(* IEC 61131-3 sources: TSA-FMICS22/benchmark/PLCopen_safety/examples, 5 files *)

(* ---- 4.1.DiagnosticsConcept.st ---- *)
PROGRAM DiagnosticsConcept
VAR_INPUT
    S1SEStopIn1 : SAFEBOOL;
    S1SEStopIn2 : SAFEBOOL;
    S2SESPEIn : SAFEBOOL;
    S0Reset : BOOL;
    S3DriveReset : BOOL;
    AxisD1 : INT;
    InputDevice1active : BOOL;
    InputDevice2active : BOOL;
    InternalAcknowledge: BOOL;
END_VAR
VAR
    SEStopOut : SAFEBOOL;
    SFEquivalent1 : SFEquivalent;
    SFEmergencyStop1 : SFEmergencyStop;
    SFESPE1 : SFESPE;
    SFSafeStop11 : SFSafeStop;
END_VAR
VAR_OUTPUT
    ErrorEquiv1 : BOOL;
    DiagEquiv1 : WORD;
    ErrorEStop1 : BOOL;
    DiagEStop1 : WORD;
    ErrorESPE1 : BOOL;
    DiagESPE1 : WORD;
    ErrorSafeStop1 : BOOL;
    DiagSafeStop1 : WORD;
    SStopped : BOOL;
END_VAR
SFEquivalent1(Activate:=InputDevice1active, SChannelA:=S1SEStopIn1, SChannelB:=S1SEStopIn2, DiscrepancyTime:=T#10ms);
SFEmergencyStop1(Activate:=SFEquivalent1.Ready, SEStopIn:=SFEquivalent1.SEquivalentOut, SStartReset:=FALSE, SAutoReset:=FALSE, Reset:=S0Reset);
SFESPE1(Activate:=InputDevice2active, SESPEIn:=S2SESPEIn, SStartReset:=FALSE, SAutoReset:=FALSE, Reset:=S0Reset);
SFSafeStop11(Activate:=SFEmergencyStop1.Ready AND SFESPE1.Ready, SStopIn:=SEStopOut AND SFESPE1.SESPEOut, AxisID:=AxisD1, MonitoringTime:=T#100ms, Reset:=S3DriveReset, Acknowledge := InternalAcknowledge);
SEStopOut := SFEmergencyStop1.SEStopOut;
ErrorEquiv1 := SFEquivalent1.Error;
DiagEquiv1 := SFEquivalent1.DiagCode;
ErrorEStop1 := SFEmergencyStop1.Error;
DiagEStop1 := SFEmergencyStop1.DiagCode;
ErrorESPE1 := SFESPE1.Error;
DiagESPE1 := SFESPE1.DiagCode;
ErrorSafeStop1 := SFSafeStop11.Error;
DiagSafeStop1 := SFSafeStop11.DiagCode;
SStopped := SFSafeStop11.SStopped;
END_PROGRAM

FUNCTION_BLOCK SFEquivalent
VAR_INPUT
    Activate : BOOL;
    SChannelA : BOOL;
    SChannelB : BOOL;
    DiscrepancyTime : TIME;
END_VAR
VAR
    Timer : TON;
END_VAR
VAR_OUTPUT
    Ready : BOOL;
	SEquivalentOut : BOOL;
	Error : BOOL;
	DiagCode : WORD;
END_VAR

IF NOT Activate THEN
    DiagCode := 16#0000;
ELSE
    CASE DiagCode OF
    16#0000:
        IF Activate THEN
            DiagCode := 16#8001;
        END_IF;
    16#8001:
        IF SChannelA AND NOT SChannelB THEN
            DiagCode := 16#8004;
        ELSIF SChannelB AND NOT SChannelA THEN
            DiagCode := 16#8014;
        ELSIF SChannelA AND SChannelB THEN
            DiagCode := 16#8000;
        END_IF;
    16#8004:
        IF Timer.Q THEN
            DiagCode := 16#C001;
        ELSIF NOT SChannelA THEN
            DiagCode := 16#8001;
        ELSIF SChannelB THEN
            DiagCode := 16#8000;
        END_IF;
    16#C001,
    16#C002:
        IF NOT SChannelA AND NOT SChannelB THEN
            DiagCode := 16#8001;
        END_IF;
    16#8014:
        IF Timer.Q THEN
            DiagCode := 16#C002;
        ELSIF NOT SChannelB THEN
            DiagCode := 16#8001;
        ELSIF SChannelA THEN
            DiagCode := 16#8000;
        END_IF;
    16#C003:
        IF NOT SChannelA AND NOT SChannelB THEN
            DiagCode := 16#8001;
        END_IF;
    16#8005:
        IF Timer.Q THEN
            DiagCode := 16#C003;
        ELSIF NOT SChannelA AND NOT SChannelB THEN
            DiagCode := 16#8001;
        END_IF;
    16#8000:
        IF SChannelA XOR SChannelB THEN
            DiagCode := 16#8005;
        ELSIF NOT SChannelA AND NOT SChannelB THEN
            DiagCode := 16#8001;
        END_IF;
    END_CASE;
END_IF;

CASE DiagCode OF
16#0000:
    Timer(IN:=FALSE, PT:=DiscrepancyTime);
    Ready := FALSE;
    Error := FALSE;
    SEquivalentOut:= FALSE;
16#8000:
    Timer(IN:=FALSE, PT:=DiscrepancyTime);
    Ready := TRUE;
    Error := FALSE;
    SEquivalentOut := TRUE;
16#8001:
    Timer(IN:=FALSE, PT:=DiscrepancyTime);
    Ready := TRUE;
    Error := FALSE;
    SEquivalentOut:= FALSE;
16#8004,
16#8014,
16#8005:
	Timer(IN:=TRUE, PT:=DiscrepancyTime);
    Ready := TRUE;
    Error := FALSE;
    SEquivalentOut:= FALSE;
16#C001,
16#C002,
16#C003:
    Timer(IN:=FALSE, PT:=DiscrepancyTime);
    Ready := TRUE;
    Error := TRUE;
    SEquivalentOut:= FALSE;
END_CASE;
END_FUNCTION_BLOCK

FUNCTION_BLOCK SFEmergencyStop
VAR_INPUT
    Activate : BOOL;
    SEStopIn : BOOL;
    SStartReset : BOOL;
    SAutoReset : BOOL;
    Reset : BOOL;
END_VAR
VAR
    RTRIGatReset : RTRIG;
END_VAR
VAR_OUTPUT
    Ready : BOOL;
    SEStopOut : BOOL;
    Error : BOOL;
    DiagCode : WORD;
END_VAR
RTRIGatReset(CLK:=Reset);
IF NOT Activate THEN
    DiagCode := 16#0000;
ELSE
    CASE DiagCode OF
    16#0000:
        IF Activate THEN
            DiagCode := 16#8001;
        END_IF;
    16#8001:
        IF NOT SStartReset THEN
            DiagCode := 16#8002;
        ELSIF SStartReset AND NOT SEStopIn THEN
            DiagCode := 16#8004;
        ELSIF SEStopIn AND SStartReset THEN
            DiagCode := 16#8000;
        END_IF;
    16#8002:
        IF SEStopIn THEN
            DiagCode := 16#8003;
        END_IF;
    16#8003:
        IF Reset AND NOT RTRIGatReset.Q THEN
            DiagCode := 16#C001;
        ELSIF NOT SEStopIn THEN
            DiagCode := 16#8002;
        ELSIF RTRIGatReset.Q THEN
            DiagCode := 16#8000;
        END_IF;
    16#C001:
        IF NOT Reset THEN
            DiagCode := 16#8003;
        END_IF;
    16#8004:
        IF SEStopIn AND NOT SAutoReset THEN
            DiagCode := 16#8005;
        ELSIF SEStopIn AND SAutoReset THEN
            DiagCode := 16#8000;
        END_IF;
    16#8005:
        IF Reset AND NOT RTRIGatReset.Q THEN
            DiagCode := 16#C002;
        ELSIF NOT SEStopIn THEN
            DiagCode := 16#8004;
        ELSIF RTRIGatReset.Q OR SAutoReset THEN
            DiagCode := 16#8000;
        END_IF;
    16#C002:
        IF NOT Reset THEN
            DiagCode := 16#8005;
        END_IF;
    16#8000:
        IF NOT SEStopIn THEN
            DiagCode := 16#8004;
        END_IF;
    END_CASE;
END_IF;
CASE DiagCode OF
16#0000:
    Ready := FALSE;
    Error := FALSE;
    SEStopOut := FALSE;
16#8001:
    Ready := TRUE;
    Error := FALSE;
    SEStopOut := FALSE;
16#8002:
    Ready := TRUE;
    Error := FALSE;
    SEStopOut := FALSE;
16#8003:
    Ready := TRUE;
    Error := FALSE;
    SEStopOut := FALSE;
16#C001:
    Ready := TRUE;
    Error := TRUE;
    SEStopOut := FALSE;
16#8004:
    Ready := TRUE;
    Error := FALSE;
    SEStopOut := FALSE;
16#8005:
    Ready := TRUE;
    Error := FALSE;
    SEStopOut := FALSE;
16#C002:
    Ready := TRUE;
    Error := TRUE;
    SEStopOut := FALSE;
16#8000:
    Ready := TRUE;
    Error := FALSE;
    SEStopOut := TRUE;
END_CASE;
END_FUNCTION_BLOCK

FUNCTION_BLOCK SFESPE
VAR_INPUT
    Activate : BOOL;
    SESPEIn : BOOL;
    SStartReset : BOOL;
    SAutoReset : BOOL;
    Reset : BOOL;
END_VAR
VAR
    RTRIGatReset : RTRIG;
END_VAR
VAR_OUTPUT
    Ready : BOOL;
    SESPEOut : BOOL;
    Error : BOOL;
    DiagCode : WORD;
END_VAR
RTRIGatReset(CLK:=Reset);
IF NOT Activate THEN
    DiagCode := 16#0000;
ELSE
    CASE DiagCode OF
    16#0000:
        IF Activate THEN
            DiagCode := 16#8001;
        END_IF;
    16#8001:
        IF NOT SStartReset THEN
            DiagCode := 16#8002;
        ELSIF SStartReset AND NOT SESPEIn THEN
            DiagCode := 16#8004;
        ELSIF SESPEIn AND SStartReset THEN
            DiagCode := 16#8000;
        END_IF;
    16#8002:
        IF SESPEIn THEN
            DiagCode := 16#8003;
        END_IF;
    16#8003:
        IF Reset AND NOT RTRIGatReset.Q THEN
            DiagCode := 16#C001;
        ELSIF NOT SESPEIn THEN
            DiagCode := 16#8002;
        ELSIF RTRIGatReset.Q THEN
            DiagCode := 16#8000;
        END_IF;
    16#C001:
        IF NOT Reset THEN
            DiagCode := 16#8003;
        END_IF;
    16#8004:
        IF SESPEIn AND NOT SAutoReset THEN
            DiagCode := 16#8005;
        ELSIF SESPEIn AND SAutoReset THEN
            DiagCode := 16#8000;
        END_IF;
    16#8005:
        IF Reset AND NOT RTRIGatReset.Q THEN
            DiagCode := 16#C002;
        ELSIF NOT SESPEIn THEN
            DiagCode := 16#8004;
        ELSIF RTRIGatReset.Q OR SAutoReset THEN
            DiagCode := 16#8000;
        END_IF;
    16#C002:
        IF NOT Reset THEN
            DiagCode := 16#8005;
        END_IF;
    16#8000:
        IF NOT SESPEIn THEN
            DiagCode := 16#8004;
        END_IF;
    END_CASE;
END_IF;
CASE DiagCode OF
16#0000:
    Ready := FALSE;
    Error := FALSE;
    SESPEOut := FALSE;
16#8001:
    Ready := TRUE;
    Error := FALSE;
    SESPEOut := FALSE;
16#8002:
    Ready := TRUE;
    Error := FALSE;
    SESPEOut := FALSE;
16#8003:
    Ready := TRUE;
    Error := FALSE;
    SESPEOut := FALSE;
16#C001:
    Ready := TRUE;
    Error := TRUE;
    SESPEOut := FALSE;
16#8004:
    Ready := TRUE;
    Error := FALSE;
    SESPEOut := FALSE;
16#8005:
    Ready := TRUE;
    Error := FALSE;
    SESPEOut := FALSE;
16#C002:
    Ready := TRUE;
    Error := TRUE;
    SESPEOut := FALSE;
16#8000:
    Ready := TRUE;
    Error := FALSE;
    SESPEOut := TRUE;
END_CASE;
END_FUNCTION_BLOCK

FUNCTION_BLOCK SFSafeStop
VAR_INPUT
    Activate : BOOL;
    SStopIn : SAFEBOOL;
    AxisID : INT;
    MonitoringTime : TIME;
    Reset : BOOL;
    Acknowledge : BOOL;      (* This is an internal input *)
END_VAR
VAR
    Timer : TON;
    RTRIGatReset : RTRIG;
END_VAR
VAR_OUTPUT
    Ready : BOOL;
    SStopped : SAFEBOOL;
    Error : BOOL;
    DiagCode : WORD:=16#0000;
END_VAR
RTRIGatReset(CLK:=Reset);
IF NOT Activate THEN
    DiagCode := 16#0000;
ELSE
    Timer(IN:=Activate AND NOT SStopIn, PT:=MonitoringTime);
    CASE DiagCode OF
    16#0000:
        IF Activate THEN
            DiagCode := 16#8001;
        END_IF;
    16#8000:
        IF NOT Acknowledge THEN
            DiagCode := 16#C002;
        ELSIF SStopIn THEN
            DiagCode := 16#8012;
        END_IF;
    16#8001:
        IF RTRIGatReset.Q AND NOT Acknowledge THEN
            DiagCode := 16#8002;
        ELSIF RTRIGatReset.Q AND Acknowledge THEN
            DiagCode := 16#8012;
        END_IF;
    16#8002:
        IF NOT SStopIn THEN
            DiagCode := 16#8003;
        ELSIF Acknowledge THEN
            DiagCode := 16#8012;
        END_IF;
    16#8003:
        IF Timer.Q THEN
            DiagCode := 16#C003;
        ELSIF SStopIn THEN
            DiagCode := 16#8012;
        ELSIF Acknowledge THEN
            DiagCode := 16#8000;
        END_IF;
    16#8005:
        IF SStopIn THEN
            DiagCode := 16#8012;
        END_IF;
    16#8012:
        IF NOT Acknowledge THEN
            DiagCode := 16#8002;
        ELSIF NOT SStopIn THEN
            DiagCode := 16#8003;
        ELSIF Acknowledge THEN
            DiagCode := 16#8000;
        END_IF;
    16#C002:
        IF Reset AND NOT RTRIGatReset.Q THEN
            DiagCode := 16#C004;
        ELSIF RTRIGatReset.Q THEN
            DiagCode := 16#8005;
        END_IF;
    16#C003:
        IF Reset AND NOT RTRIGatReset.Q THEN
            DiagCode := 16#C005;
        ELSIF RTRIGatReset.Q THEN
            DiagCode := 16#8005;
        END_IF;
    16#C004:
        IF NOT Reset THEN
            DiagCode := 16#C002;
        END_IF;
    16#C005:
        IF NOT Reset THEN
            DiagCode := 16#C003;
        END_IF;
    END_CASE;
END_IF;
CASE DiagCode OF
16#0000:
    Ready := FALSE;
    SStopped := FALSE;
    Error := FALSE;
16#8000:
    Ready := TRUE;
    SStopped := TRUE;
    Error := FALSE;
16#8001,
16#8002,
16#8003,
16#8005,
16#8012:
    Ready := TRUE;
    SStopped := FALSE;
    Error := FALSE;
16#C002,
16#C003,
16#C004,
16#C005:
    Ready := TRUE;
    SStopped := FALSE;
    Error := TRUE;
END_CASE;
END_FUNCTION_BLOCK

FUNCTION_BLOCK RTRIG
VAR_INPUT
    CLK : BOOL;
END_VAR
VAR
    M : BOOL;
END_VAR
VAR_OUTPUT
    Q : BOOL;
END_VAR
    Q := CLK AND NOT M;
    M := CLK;
END_FUNCTION_BLOCK

FUNCTION_BLOCK TON
VAR_INPUT
    IN : BOOL;
    PT : TIME;
END_VAR
VAR
    running : BOOL;
END_VAR
VAR_TEMP
    timeout : BOOL;
END_VAR
VAR_OUTPUT
    Q : BOOL;
    ET : TIME;
END_VAR
timeout := NONDETERMINISTIC_BOOL();
IF NOT IN THEN
    Q := FALSE;
    running := FALSE;
ELSIF NOT running AND NOT Q THEN
    running := TRUE;
ELSIF running AND NOT Q THEN
    Q := timeout;
    running := NOT Q;
END_IF;
ET := NONDETERMINISTIC_TIME();
END_FUNCTION_BLOCK

(* ---- 4.2.SafeMotion.st ---- *)
PROGRAM SafeMotion
VAR_INPUT
    S1SEStopIn : SAFEBOOL;
    S2SMode0 : SAFEBOOL;
    S2SMode1 : SAFEBOOL;
    S4SEnableSwitchCh1 : SAFEBOOL;
    S4SEnableSwitchCh2 : SAFEBOOL;
    S5SGuardSwitch1 : SAFEBOOL;
    S6SGuardSwitch2 : SAFEBOOL;
    S7SGuardLock : SAFEBOOL;
    S0Reset : BOOL;
    S8UnlockGuard : BOOL;
    SFSafeStop11ACK: BOOL;
    SFSafeStop12ACK: BOOL;
    SFSLS1ACK: BOOL;
    SFSLS2ACK: BOOL;
END_VAR
VAR_OUTPUT
    SUnlockGuardK1 : SAFEBOOL;
END_VAR
VAR
    SSafeStopAxis1 : SAFEBOOL;
    SSafeStopAxis2 : SAFEBOOL;
    SSafeMoveAxis1 : SAFEBOOL;
    SSafeMoveAxis2 : SAFEBOOL;
    SSafetyActive : SAFEBOOL;
    SModeAutoActive : SAFEBOOL;
    SModeSetSel : SAFEBOOL;
    SSLSEnable : SAFEBOOL;
    SGuardLocked : SAFEBOOL;
    SFEmergencyStop1 : SFEmergencyStop;
    SFSafeStop11 : SFSafeStop;
    SFSafeStop12 : SFSafeStop;
    SFModeSelector1 : SFModeSelector;
    SFGuardMonitoring1 : SFGuardMonitoring;
    SFGuardLocking1 : SFGuardLocking;
    SFEnableSwitch1 : SFEnableSwitch;
    SFSafelyLimitedSpeed1 : SFSafelyLimitSpeed;
    SFSafelyLimitedSpeed2 : SFSafelyLimitSpeed;
END_VAR

SFEmergencyStop1(Activate:=TRUE, SEStopIn:=S1SEStopIn, SStartReset:=FALSE, SAutoReset:=FALSE, Reset:=S0Reset);
SFSafeStop11(Activate:=TRUE, SStopIn:=SFEmergencyStop1.SEStopOut, AxisID:=1, MonitoringTime:=T#1s, Reset:=S0Reset, Acknowledge:=SFSafeStop11ACK);
SSafeStopAxis1 := SFSafeStop11.SStopped;
SFSafeStop12(Activate:=TRUE, SStopIn:=SFEmergencyStop1.SEStopOut, AxisID:=2, MonitoringTime:=T#1s, Reset:=S0Reset, Acknowledge:=SFSafeStop12ACK);
SSafeStopAxis2 := SFSafeStop12.SStopped;

SFModeSelector1(Activate:=TRUE, SMode0:=S2SMode0, SMode1:=S2SMode1, SMode2:=FALSE, SMode3:=FALSE, SMode4:=FALSE, SMode5:=FALSE, SMode6:=FALSE, SMode7:=FALSE, SUnlock:=TRUE, SSetMode:=FALSE,
 AutoSetMode:=TRUE, ModeMonitorTime:=T#50ms, Reset:=S0Reset);
SModeSetSel := SFModeSelector1.SMode1Sel;
SModeAutoActive := SFModeSelector1.SMode0Sel AND SGuardLocked;

SFGuardMonitoring1(Activate:=TRUE, SGuardSwitch1:=S5SGuardSwitch1, SGuardSwitch2:=S6SGuardSwitch2, DiscrepancyTime:=T#50ms, SStartReset:=FALSE, SAutoReset:=FALSE, Reset:=S0Reset);
SSafetyActive := (SSafeStopAxis1 AND SSafeStopAxis2) OR (SFSafelyLimitedSpeed1.SSafetyActive AND SFSafelyLimitedSpeed2.SSafetyActive);

SFGuardLocking1(Activate:=TRUE, SGuardMonitoring:=SFGuardMonitoring1.SGuardMonitoring, SSafetyActive:=SSafetyActive, SGuardLock:=S7SGuardLock, UnlockRequest:=S8UnlockGuard, SStartReset:=FALSE,
 SAutoReset:=FALSE, Reset:=S0Reset);
SGuardLocked := SFGuardLocking1.SGuardLocked;
SUnlockGuardK1 := SFGuardLocking1.SUnlockGuard;

SFEnableSwitch1(Activate:=TRUE, SSafetyActive:=SSafetyActive AND SModeSetSel, SEnableSwitchCh1:=S4SEnableSwitchCh1, SEnableSwitchCh2:=S4SEnableSwitchCh2, SAutoReset:=FALSE, Reset:=S0Reset);
SSLSEnable := SFEnableSwitch1.SEnableSwitchOut;

SFSafelyLimitedSpeed1(Activate:=TRUE, SOpMode:=SFModeSelector1.SMode0Sel AND SGuardLocked, SEnabled:=SSLSEnable, AxisID:=1, MonitoringTime:=T#1s, Reset:=S0Reset, Acknowledge:=SFSLS1ACK);
SSafeMoveAxis1 := SFSafelyLimitedSpeed1.SSafetyActive;

SFSafelyLimitedSpeed2(Activate:=TRUE, SOpMode:=SFModeSelector1.SMode0Sel AND SGuardLocked, SEnabled:=SSLSEnable, AxisID:=2, MonitoringTime:=T#1s, Reset:=S0Reset, Acknowledge:=SFSLS2ACK);
SSafeMoveAxis2 := SFSafelyLimitedSpeed2.SSafetyActive;
END_PROGRAM

FUNCTION_BLOCK SFEmergencyStop
VAR_INPUT
    Activate : BOOL;
    SEStopIn : BOOL;
    SStartReset : BOOL;
    SAutoReset : BOOL;
    Reset : BOOL;
END_VAR
VAR
    RTRIGatReset : RTRIG;
END_VAR
VAR_OUTPUT
    Ready : BOOL;
    SEStopOut : BOOL;
    Error : BOOL;
    DiagCode : WORD;
END_VAR
RTRIGatReset(CLK:=Reset);
IF NOT Activate THEN
    DiagCode := 16#0000;
ELSE
    CASE DiagCode OF
    16#0000:
        IF Activate THEN
            DiagCode := 16#8001;
        END_IF;
    16#8001:
        IF NOT SStartReset THEN
            DiagCode := 16#8002;
        ELSIF SStartReset AND NOT SEStopIn THEN
            DiagCode := 16#8004;
        ELSIF SEStopIn AND SStartReset THEN
            DiagCode := 16#8000;
        END_IF;
    16#8002:
        IF SEStopIn THEN
            DiagCode := 16#8003;
        END_IF;
    16#8003:
        IF Reset AND NOT RTRIGatReset.Q THEN
            DiagCode := 16#C001;
        ELSIF NOT SEStopIn THEN
            DiagCode := 16#8002;
        ELSIF RTRIGatReset.Q THEN
            DiagCode := 16#8000;
        END_IF;
    16#C001:
        IF NOT Reset THEN
            DiagCode := 16#8003;
        END_IF;
    16#8004:
        IF SEStopIn AND NOT SAutoReset THEN
            DiagCode := 16#8005;
        ELSIF SEStopIn AND SAutoReset THEN
            DiagCode := 16#8000;
        END_IF;
    16#8005:
        IF Reset AND NOT RTRIGatReset.Q THEN
            DiagCode := 16#C002;
        ELSIF NOT SEStopIn THEN
            DiagCode := 16#8004;
        ELSIF RTRIGatReset.Q OR SAutoReset THEN
            DiagCode := 16#8000;
        END_IF;
    16#C002:
        IF NOT Reset THEN
            DiagCode := 16#8005;
        END_IF;
    16#8000:
        IF NOT SEStopIn THEN
            DiagCode := 16#8004;
        END_IF;
    END_CASE;
END_IF;
CASE DiagCode OF
16#0000:
    Ready := FALSE;
    Error := FALSE;
    SEStopOut := FALSE;
16#8001:
    Ready := TRUE;
    Error := FALSE;
    SEStopOut := FALSE;
16#8002:
    Ready := TRUE;
    Error := FALSE;
    SEStopOut := FALSE;
16#8003:
    Ready := TRUE;
    Error := FALSE;
    SEStopOut := FALSE;
16#C001:
    Ready := TRUE;
    Error := TRUE;
    SEStopOut := FALSE;
16#8004:
    Ready := TRUE;
    Error := FALSE;
    SEStopOut := FALSE;
16#8005:
    Ready := TRUE;
    Error := FALSE;
    SEStopOut := FALSE;
16#C002:
    Ready := TRUE;
    Error := TRUE;
    SEStopOut := FALSE;
16#8000:
    Ready := TRUE;
    Error := FALSE;
    SEStopOut := TRUE;
END_CASE;
END_FUNCTION_BLOCK

FUNCTION_BLOCK SFSafeStop
VAR_INPUT
    Activate : BOOL;
    SStopIn : SAFEBOOL;
    AxisID : INT;
    MonitoringTime : TIME;
    Reset : BOOL;
    Acknowledge : BOOL;      (* This is an internal input *)
END_VAR
VAR
    Timer : TON;
    RTRIGatReset : RTRIG;
END_VAR
VAR_OUTPUT
    Ready : BOOL;
    SStopped : SAFEBOOL;
    Error : BOOL;
    DiagCode : WORD:=16#0000;
END_VAR
RTRIGatReset(CLK:=Reset);
IF NOT Activate THEN
    DiagCode := 16#0000;
ELSE
    Timer(IN:=Activate AND NOT SStopIn, PT:=MonitoringTime);
    CASE DiagCode OF
    16#0000:
        IF Activate THEN
            DiagCode := 16#8001;
        END_IF;
    16#8000:
        IF NOT Acknowledge THEN
            DiagCode := 16#C002;
        ELSIF SStopIn THEN
            DiagCode := 16#8012;
        END_IF;
    16#8001:
        IF RTRIGatReset.Q AND NOT Acknowledge THEN
            DiagCode := 16#8002;
        ELSIF RTRIGatReset.Q AND Acknowledge THEN
            DiagCode := 16#8012;
        END_IF;
    16#8002:
        IF NOT SStopIn THEN
            DiagCode := 16#8003;
        ELSIF Acknowledge THEN
            DiagCode := 16#8012;
        END_IF;
    16#8003:
        IF Timer.Q THEN
            DiagCode := 16#C003;
        ELSIF SStopIn THEN
            DiagCode := 16#8012;
        ELSIF Acknowledge THEN
            DiagCode := 16#8000;
        END_IF;
    16#8005:
        IF SStopIn THEN
            DiagCode := 16#8012;
        END_IF;
    16#8012:
        IF NOT Acknowledge THEN
            DiagCode := 16#8002;
        ELSIF NOT SStopIn THEN
            DiagCode := 16#8003;
        ELSIF Acknowledge THEN
            DiagCode := 16#8000;
        END_IF;
    16#C002:
        IF Reset AND NOT RTRIGatReset.Q THEN
            DiagCode := 16#C004;
        ELSIF RTRIGatReset.Q THEN
            DiagCode := 16#8005;
        END_IF;
    16#C003:
        IF Reset AND NOT RTRIGatReset.Q THEN
            DiagCode := 16#C005;
        ELSIF RTRIGatReset.Q THEN
            DiagCode := 16#8005;
        END_IF;
    16#C004:
        IF NOT Reset THEN
            DiagCode := 16#C002;
        END_IF;
    16#C005:
        IF NOT Reset THEN
            DiagCode := 16#C003;
        END_IF;
    END_CASE;
END_IF;
CASE DiagCode OF
16#0000:
    Ready := FALSE;
    SStopped := FALSE;
    Error := FALSE;
16#8000:
    Ready := TRUE;
    SStopped := TRUE;
    Error := FALSE;
16#8001,
16#8002,
16#8003,
16#8005,
16#8012:
    Ready := TRUE;
    SStopped := FALSE;
    Error := FALSE;
16#C002,
16#C003,
16#C004,
16#C005:
    Ready := TRUE;
    SStopped := FALSE;
    Error := TRUE;
END_CASE;
END_FUNCTION_BLOCK

FUNCTION_BLOCK SFModeSelector
VAR_INPUT
    Activate : BOOL;
    SMode0 : BOOL;
    SMode1 : BOOL;
    SMode2 : BOOL;
    SMode3 : BOOL;
    SMode4 : BOOL;
    SMode5 : BOOL;
    SMode6 : BOOL;
    SMode7 : BOOL;
    SUnlock : BOOL;
    SSetMode : BOOL;
    AutoSetMode : BOOL;
    ModeMonitorTime : TIME;
    Reset : BOOL;
END_VAR
VAR
    Timer : TON;
    RTRIGatReset: RTRIG;
    RTRIGatSetMode: RTRIG;
    FTRIGatModeSel0: FTRIG;
    RTRIGatModeSel0: RTRIG;
    fallingEdgeDetected : BOOL;
END_VAR
VAR_TEMP
    Error1 : BOOL;
    Error2 : BOOL;
END_VAR
VAR_OUTPUT
    Ready : BOOL;
    SMode0Sel : BOOL;
    SMode1Sel : BOOL;
    SMode2Sel : BOOL;
    SMode3Sel : BOOL;
    SMode4Sel : BOOL;
    SMode5Sel : BOOL;
    SMode6Sel : BOOL;
    SMode7Sel : BOOL;
    SAnyModeSel : BOOL;
    Error : BOOL;
    DiagCode : WORD;
END_VAR
RTRIGatReset(CLK:=Reset);
RTRIGatSetMode(CLK:=SSetMode);
IF NOT Activate THEN
    DiagCode := 16#0000;
ELSE
    IF (SMode0 + SMode1 + SMode2 + SMode3 + SMode4 + SMode5 + SMode6 + SMode7 > 1) THEN
        Error1 := true;
    ELSE
        Error1 := false;
    END_IF;
    CASE DiagCode OF
    16#0000:
        IF Activate THEN
            DiagCode := 16#8005;
        END_IF;
    16#8005:
        IF (NOT SMode0 AND NOT SMode1 AND NOT SMode2 AND NOT SMode3 AND NOT SMode4 AND NOT SMode5 AND NOT SMode6 AND NOT SMode7) THEN
            FTRIGatModeSel0(CLK:=false);
            RTRIGatModeSel0(CLK:=false);
        ELSE
            FTRIGatModeSel0(CLK:=true);
            RTRIGatModeSel0(CLK:=true);
        END_IF;
        IF FTRIGatModeSel0.Q THEN
            fallingEdgeDetected := TRUE;
        END_IF;
        IF fallingEdgeDetected THEN
            Timer(IN:=TRUE, PT:=ModeMonitorTime);
        ELSIF RTRIGatModeSel0.Q THEN
            Timer(IN:=FALSE, PT:=ModeMonitorTime);
            fallingEdgeDetected := FALSE;
        END_IF;
        Error2 := Timer.Q;
        IF Error1 THEN
            DiagCode := 16#C001;
        ELSIF Error2 THEN
            DiagCode := 16#C002;
        ELSIF ((AutoSetMode OR RTRIGatSetMode.Q) AND SUnlock AND (SMode0 + SMode1 + SMode2 + SMode3 + SMode4 + SMode5 + SMode6 + SMode7 = 1)) THEN
            DiagCode := 16#8000;
        END_IF;
    16#8000:
        IF Error1 THEN
            DiagCode := 16#C001;
        ELSIF (SMode0 <> SMode0Sel OR SMode1 <> SMode1Sel OR SMode2 <> SMode2Sel OR SMode3 <> SMode3Sel
              OR SMode4 <> SMode4Sel OR SMode5 <> SMode5Sel OR SMode6 <> SMode6Sel OR SMode7 <> SMode7Sel) THEN
            DiagCode := 16#8005;
            fallingEdgeDetected := FALSE;
        ELSIF (NOT SUnlock) THEN
            DiagCode := 16#8004;
        END_IF;
    16#8004:
        IF SUnlock THEN
            DiagCode := 16#8000;
        END_IF;
    16#C001:
        IF Reset AND NOT RTRIGatReset.Q THEN
            DiagCode := 16#C003;
        ELSIF RTRIGatReset.Q THEN
            DiagCode := 16#8005;
            fallingEdgeDetected := FALSE;
        END_IF;
    16#C002:
        IF Reset AND NOT RTRIGatReset.Q THEN
            DiagCode := 16#C004;
        ELSIF RTRIGatReset.Q THEN
            DiagCode := 16#8005;
            fallingEdgeDetected := FALSE;
        END_IF;
    16#C003:
        IF (NOT Reset) THEN
            DiagCode := 16#C001;
        END_IF;
    16#C004:
        IF (NOT Reset) THEN
            DiagCode := 16#C002;
        END_IF;
    END_CASE;
END_IF;

CASE DiagCode OF
16#0000:
    Ready := false;
    SMode0Sel := false;
    SMode1Sel := false;
    SMode2Sel := false;
    SMode3Sel := false;
    SMode4Sel := false;
    SMode5Sel := false;
    SMode6Sel := false;
    SMode7Sel := false;
    SAnyModeSel := false;
    Error := false;
16#8005:
    Ready := true;
    SMode0Sel := false;
    SMode1Sel := false;
    SMode2Sel := false;
    SMode3Sel := false;
    SMode4Sel := false;
    SMode5Sel := false;
    SMode6Sel := false;
    SMode7Sel := false;
    SAnyModeSel := false;
    Error := false;
16#8000:
    Ready := true;
    SMode0Sel := SMode0;
    SMode1Sel := SMode1;
    SMode2Sel := SMode2;
    SMode3Sel := SMode3;
    SMode4Sel := SMode4;
    SMode5Sel := SMode5;
    SMode6Sel := SMode6;
    SMode7Sel := SMode7;
    SAnyModeSel := true;
    Error := false;
16#8004:
    Ready := true;
    SAnyModeSel := true;
    Error := false;
16#C001,
16#C002,
16#C003,
16#C004:
    Ready := true;
    SMode0Sel := false;
    SMode1Sel := false;
    SMode2Sel := false;
    SMode3Sel := false;
    SMode4Sel := false;
    SMode5Sel := false;
    SMode6Sel := false;
    SMode7Sel := false;
    SAnyModeSel := false;
    Error := true;
END_CASE;
IF (DiagCode <> 16#8005) THEN
    Timer(IN:=FALSE, PT:=ModeMonitorTime);
END_IF;
END_FUNCTION_BLOCK

FUNCTION_BLOCK SFGuardMonitoring
VAR_INPUT
    Activate : BOOL := FALSE;
    SGuardSwitch1 : SAFEBOOL := FALSE;
    SGuardSwitch2 : SAFEBOOL := FALSE;
    DiscrepancyTime : TIME := T#0s;
    SStartReset : SAFEBOOL := FALSE;
    SAutoReset : SAFEBOOL := FALSE;
    Reset : BOOL := FALSE;
END_VAR
VAR
    Timer : TON;
    RTRIGatReset : RTRIG;
END_VAR
VAR_OUTPUT
    Ready : BOOL := FALSE;
    SGuardMonitoring : BOOL := FALSE;
    Error : BOOL := FALSE;
    DiagCode : WORD := 16#0000;
END_VAR
RTRIGatReset(CLK:=Reset);
IF NOT Activate THEN
    DiagCode := 16#0000;
ELSE
    CASE DiagCode OF
    16#0000:
        IF Activate THEN
            DiagCode := 16#8001;
        END_IF;
    16#8001:
        IF NOT SGuardSwitch1 OR NOT SGuardSwitch2 THEN
            DiagCode := 16#8002;
        ELSIF SGuardSwitch1 AND SGuardSwitch2 AND NOT SStartReset THEN
            DiagCode := 16#8003;
        ELSIF SGuardSwitch1 AND SGuardSwitch2 AND SStartReset THEN
            DiagCode := 16#8000;
        END_IF;
    16#8002:
        IF NOT SGuardSwitch1 AND NOT SGuardSwitch2 THEN
            DiagCode := 16#8012;
        END_IF;
    16#8003:
        IF Reset AND NOT RTRIGatReset.Q THEN
            DiagCode := 16#C001;
        ELSIF NOT SGuardSwitch1 OR NOT SGuardSwitch2 THEN
            DiagCode := 16#8002;
        ELSIF RTRIGatReset.Q THEN
            DiagCode := 16#8000;
        END_IF;
    16#8012:
        IF SGuardSwitch1 THEN
            DiagCode := 16#8004;
        ELSIF SGuardSwitch2 THEN
            DiagCode := 16#8014;
        END_IF;
    16#8004:
        IF Timer.Q THEN
            DiagCode := 16#C011;
        ELSIF NOT SGuardSwitch1 THEN
            DiagCode := 16#8002;
        ELSIF SGuardSwitch2 THEN
            DiagCode := 16#8005;
        END_IF;
    16#8014:
        IF Timer.Q THEN
            DiagCode := 16#C012;
        ELSIF NOT SGuardSwitch2 THEN
            DiagCode := 16#8002;
        ELSIF SGuardSwitch1 THEN
            DiagCode := 16#8005;
        END_IF;
    16#8005:
        IF NOT SGuardSwitch1 OR NOT SGuardSwitch2 THEN
            DiagCode := 16#8002;
        ELSIF NOT SAutoReset THEN
            DiagCode := 16#8003;
        ELSIF SAutoReset THEN
            DiagCode := 16#8000;
        END_IF;
    16#8000:
        IF NOT SGuardSwitch1 OR NOT SGuardSwitch2 THEN
            DiagCode := 16#8002;
        END_IF;
    16#C001:
        IF NOT Reset THEN
            DiagCode := 16#8003;
        END_IF;
    16#C011:
        IF NOT SGuardSwitch1 AND NOT SGuardSwitch2 THEN
            DiagCode := 16#8012;
        END_IF;
    16#C012:
        IF NOT SGuardSwitch1 AND NOT SGuardSwitch2 THEN
            DiagCode := 16#8012;
        END_IF;
    END_CASE;
END_IF;
CASE DiagCode OF
16#0000:
    Timer(IN:=FALSE, PT:=DiscrepancyTime);
    Ready := FALSE;
    Error := FALSE;
    SGuardMonitoring := FALSE;
16#8000:
    Timer(IN:=FALSE, PT:=DiscrepancyTime);
    Ready := TRUE;
    Error := FALSE;
    SGuardMonitoring  := TRUE;
16#8001,
16#8002,
16#8003,
16#8012,
16#8005:
    Timer(IN:=FALSE, PT:=DiscrepancyTime);
    Ready := TRUE;
    Error := FALSE;
    SGuardMonitoring := FALSE;
16#8004,
16#8014:
    Timer(IN:=TRUE, PT:=DiscrepancyTime);
    Ready := TRUE;
    Error := FALSE;
    SGuardMonitoring := FALSE;
16#C001,
16#C011,
16#C012:
    Timer(IN:=FALSE, PT:=DiscrepancyTime);
    Ready := TRUE;
    Error := TRUE;
    SGuardMonitoring := FALSE;
END_CASE;
END_FUNCTION_BLOCK

FUNCTION_BLOCK SFGuardLocking
VAR_INPUT
    Activate : BOOL;
    SGuardMonitoring : SAFEBOOL;
    SSafetyActive : SAFEBOOL;
    SGuardLock : SAFEBOOL;
    UnlockRequest : BOOL;
    SStartReset : SAFEBOOL;
    SAutoReset : SAFEBOOL;
    Reset : BOOL;
END_VAR
VAR
    RTRIGatReset : RTRIG;
    RTRIGatUnlockRequest : RTRIG;
END_VAR
VAR_OUTPUT
    Ready : BOOL;
    SGuardLocked : SAFEBOOL;
    SUnlockGuard : SAFEBOOL;
    Error : BOOL;
    DiagCode : WORD;
END_VAR
RTRIGatReset(CLK:=Reset);
RTRIGatUnlockRequest(CLK:=UnlockRequest);
IF NOT Activate THEN
    DiagCode := 16#0000;
END_IF;
CASE DiagCode OF
16#0000:
    IF Activate THEN
        DiagCode := 16#8001;
    END_IF;
16#8000:
    IF NOT SGuardLock OR NOT SGuardMonitoring THEN
        DiagCode := 16#C004;
    ELSIF RTRIGatUnlockRequest.Q AND SSafetyActive THEN
        DiagCode := 16#8013;
    END_IF;
16#8001:
    IF Reset AND NOT RTRIGatReset.Q AND NOT SStartReset THEN
        DiagCode := 16#C001;
    ELSIF NOT SGuardLock OR NOT SGuardMonitoring THEN
        DiagCode := 16#8011;
    ELSIF (RTRIGatReset.Q OR SStartReset) AND SGuardMonitoring AND SGuardLock THEN
        DiagCode := 16#8000;
    END_IF;
16#8003:
    IF Reset AND NOT RTRIGatReset.Q AND NOT SAutoReset THEN
        DiagCode := 16#C003;
    ELSIF NOT SGuardMonitoring OR NOT SGuardLock THEN
        DiagCode := 16#8011;
    ELSIF RTRIGatReset.Q OR SAutoReset THEN
        DiagCode := 16#8000;
    END_IF;
16#8011:
    IF NOT SSafetyActive AND (NOT SGuardMonitoring OR NOT SGuardLock) THEN
        DiagCode := 16#C004;
    ELSIF (SSafetyActive AND UnlockRequest) OR NOT SGuardMonitoring THEN
        DiagCode := 16#8012;
    ELSIF SGuardMonitoring AND SGuardLock THEN
        DiagCode := 16#8003;
    END_IF;
16#8012:
    IF SGuardMonitoring THEN
        DiagCode := 16#8013;
    ELSIF NOT SSafetyActive AND NOT SGuardMonitoring THEN
        DiagCode := 16#C004;
    END_IF;
16#8013:
    IF NOT SGuardMonitoring THEN
        DiagCode := 16#8012;
    ELSIF NOT UnlockRequest THEN
        DiagCode := 16#8011;
    END_IF;
16#8014:
    IF Reset AND NOT RTRIGatReset.Q THEN
        DiagCode := 16#C002;
    ELSIF NOT SSafetyActive THEN
        DiagCode := 16#C004;
    ELSIF RTRIGatReset.Q THEN
        DiagCode := 16#8011;
    END_IF;
16#C001:
    IF NOT Reset THEN
        DiagCode := 16#8001;
    END_IF;
16#C002:
    IF NOT Reset THEN
        DiagCode := 16#8014;
    END_IF;
16#C003:
    IF NOT Reset THEN
        DiagCode := 16#8003;
    END_IF;
16#C004:
    IF SSafetyActive THEN
        DiagCode := 16#8014;
    END_IF;
END_CASE;
CASE DiagCode OF
16#0000:
    Ready := FALSE;
    SGuardLocked := FALSE;
    SUnlockGuard := FALSE;
    Error := FALSE;
16#8000:
    Ready := TRUE;
    SGuardLocked := TRUE;
    SUnlockGuard := FALSE;
    Error := FALSE;
16#8001,
16#8003,
16#8011,
16#8014:
    Ready := TRUE;
    SGuardLocked := FALSE;
    SUnlockGuard := FALSE;
    Error := FALSE;
16#8012,
16#8013:
    Ready := TRUE;
    SGuardLocked := FALSE;
    SUnlockGuard := TRUE;
    Error := FALSE;
16#C001,
16#C002,
16#C003,
16#C004:
    Ready := TRUE;
    SGuardLocked := FALSE;
    SUnlockGuard := FALSE;
    Error := TRUE;
END_CASE;
END_FUNCTION_BLOCK

FUNCTION_BLOCK SFEnableSwitch
VAR_INPUT
    Activate : BOOL;
    SSafetyActive : SAFEBOOL;
    SEnableSwitchCh1 : SAFEBOOL;
    SEnableSwitchCh2 : SAFEBOOL;
    SAutoReset : SAFEBOOL;
    Reset : BOOL;
END_VAR
VAR
    RTRIGatReset : RTRIG;
END_VAR
VAR_OUTPUT
    Ready : BOOL;
    SEnableSwitchOut : SAFEBOOL;
    Error : BOOL;
    DiagCode : WORD;
END_VAR
RTRIGatReset(CLK:=Reset);
IF NOT Activate THEN
    DiagCode := 16#0000;
ELSIF NOT SSafetyActive THEN
    DiagCode := 16#8004;
ELSE
    CASE DiagCode OF
    16#0000:
        IF Activate THEN
            DiagCode := 16#8004;
        END_IF;
    16#8000:
        IF (NOT (SEnableSwitchCh1 OR SEnableSwitchCh2)) OR (SEnableSwitchCh1 AND NOT SEnableSwitchCh2) THEN
            DiagCode := 16#8007;
        ELSIF NOT SEnableSwitchCh1 AND SEnableSwitchCh2 THEN
            DiagCode := 16#8006;
        END_IF;
    16#8004:
        IF SSafetyActive THEN
            DiagCode := 16#8005;
        END_IF;
    16#8005:
        IF NOT (NOT SEnableSwitchCh1 AND SEnableSwitchCh2) THEN
            DiagCode := 16#C010;
        ELSIF NOT SEnableSwitchCh1 AND SEnableSwitchCh2 THEN
            DiagCode := 16#8006;
        END_IF;
    16#8006:
        IF SEnableSwitchCh1 AND SEnableSwitchCh2 THEN
            DiagCode := 16#8000;
        ELSIF (NOT (SEnableSwitchCh1 OR SEnableSwitchCh2)) OR (SEnableSwitchCh1 AND NOT SEnableSwitchCh2) THEN
            DiagCode := 16#8007;
        END_IF;
    16#8007:
        IF SEnableSwitchCh1 AND SEnableSwitchCh2 THEN
            DiagCode := 16#C030;
        ELSIF NOT SEnableSwitchCh1 AND SEnableSwitchCh2 THEN
            DiagCode := 16#8006;
        END_IF;
    16#C001:
        IF NOT Reset THEN
            DiagCode := 16#C020;
        END_IF;
    16#C002:
        IF NOT Reset THEN
            DiagCode := 16#C040;
        END_IF;
    16#C010:
        IF NOT SEnableSwitchCh1 AND SEnableSwitchCh2 THEN
            DiagCode := 16#C020;
        END_IF;
    16#C020:
        IF NOT (NOT SEnableSwitchCh1 AND SEnableSwitchCh2) THEN
            DiagCode := 16#C010;
        ELSIF Reset AND NOT RTRIGatReset.Q AND NOT SAutoReset THEN
            DiagCode := 16#C001;
        ELSIF RTRIGatReset.Q OR SAutoReset THEN
            DiagCode := 16#8006;
        END_IF;
    16#C030:
        IF NOT (SEnableSwitchCh1 AND SEnableSwitchCh2) THEN
            DiagCode := 16#C040;
        END_IF;
    16#C040:
        IF SEnableSwitchCh1 AND SEnableSwitchCh2 THEN
            DiagCode := 16#C030;
        ELSIF Reset AND RTRIGatReset.Q AND NOT SAutoReset THEN
            DiagCode := 16#C002;
        ELSIF RTRIGatReset.Q OR SAutoReset THEN
            DiagCode := 16#8007;
        END_IF;
    END_CASE;
END_IF;

CASE DiagCode OF
16#C001,
16#C002,
16#C010,
16#C020,
16#C030,
16#C040:
    Ready := TRUE;
    SEnableSwitchOut := FALSE;
    Error := TRUE;
16#0000:
    Ready := FALSE;
    SEnableSwitchOut := FALSE;
    Error := FALSE;
16#8000:
    Ready := TRUE;
    SEnableSwitchOut := TRUE;
    Error := FALSE;
16#8004,
16#8005,
16#8006,
16#8007:
    Ready := TRUE;
    SEnableSwitchOut := FALSE;
    Error := FALSE;
END_CASE;
END_FUNCTION_BLOCK

FUNCTION_BLOCK SFSafelyLimitSpeed
VAR_INPUT
    Activate : BOOL;
    SOpMode : SAFEBOOL;
    SEnabled : SAFEBOOL;
    AxisID : INT;
    MonitoringTime : TIME;
    Reset : BOOL;
    Acknowledge : BOOL;      (* This is an internal input *)
END_VAR
VAR
    Timer: TON;
    RTRIGatReset: RTRIG;
END_VAR
VAR_OUTPUT
    Ready : BOOL;
    SSafetyActive : SAFEBOOL;
    Error : BOOL;
    DiagCode : WORD;
END_VAR
RTRIGatReset(CLK:=Reset);
IF NOT Activate THEN
    DiagCode := 16#0000;
END_IF;
Timer(IN:=Activate AND NOT SOpMode, PT:=MonitoringTime);
CASE DiagCode OF
16#0000:
    IF Activate THEN
        DiagCode := 16#8001;
    END_IF;
16#8000:
    IF NOT Acknowledge THEN
        DiagCode := 16#C002;
    ELSIF SOpMode THEN
        DiagCode := 16#8012;
    ELSIF SEnabled THEN
        DiagCode := 16#8004;
    END_IF;
16#8001:
    IF Reset AND NOT RTRIGatReset.Q THEN
        DiagCode := 16#C001;
    ELSIF RTRIGatReset.Q AND NOT Acknowledge THEN
        DiagCode := 16#8002;
    ELSIF RTRIGatReset.Q AND Acknowledge THEN
        DiagCode := 16#8012;
    END_IF;
16#8002:
    IF NOT SOpMode THEN
        DiagCode := 16#8003;
    ELSIF Acknowledge THEN
        DiagCode := 16#8012;
    END_IF;
16#8003:
    IF Timer.Q THEN
        DiagCode := 16#C003;
    ELSIF SOpMode THEN
        DiagCode := 16#8012;
    ELSIF Acknowledge AND NOT SEnabled THEN
        DiagCode := 16#8000;
    ELSIF Acknowledge AND SEnabled THEN
        DiagCode := 16#8004;
    END_IF;
16#8004:
    IF NOT Acknowledge THEN
        DiagCode := 16#C002;
    ELSIF SOpMode THEN
        DiagCode := 16#8012;
    ELSIF NOT SEnabled THEN
        DiagCode := 16#8000;
    END_IF;
16#8005:
    IF SOpMode THEN
        DiagCode := 16#8012;
    END_IF;
16#8012:
    IF NOT Acknowledge THEN
        DiagCode := 16#8002;
    ELSIF NOT SOpMode THEN
        DiagCode := 16#8003;
    END_IF;
16#C001:
    IF NOT Reset THEN
        DiagCode := 16#8001;
    END_IF;
16#C002:
    IF Reset AND NOT RTRIGatReset.Q THEN
        DiagCode := 16#C004;
    ELSIF RTRIGatReset.Q THEN
        DiagCode := 16#8005;
    END_IF;
16#C003:
    IF Reset AND NOT RTRIGatReset.Q THEN
        DiagCode := 16#C005;
    ELSIF RTRIGatReset.Q THEN
        DiagCode := 16#8005;
    END_IF;
16#C004:
    IF NOT Reset THEN
        DiagCode := 16#C002;
    END_IF;
16#C005:
    IF NOT Reset THEN
        DiagCode := 16#C003;
    END_IF;
END_CASE;
CASE DiagCode OF
16#0000:
    Ready := FALSE;
    SSafetyActive := FALSE;
    Error := FALSE;
16#8000,
16#8004:
    Ready := TRUE;
    SSafetyActive := TRUE;
    Error := FALSE;
16#8001,
16#8002,
16#8003,
16#8005,
16#8012:
    Ready := TRUE;
    SSafetyActive := FALSE;
    Error := FALSE;
16#C001,
16#C002,
16#C003,
16#C004,
16#C005:
    Ready := TRUE;
    SSafetyActive := FALSE;
    Error := TRUE;
END_CASE;
END_FUNCTION_BLOCK

FUNCTION_BLOCK TON
VAR_INPUT
    IN : BOOL;
    PT : TIME;
END_VAR
VAR
    running : BOOL;
END_VAR
VAR_TEMP
    timeout : BOOL;
END_VAR
VAR_OUTPUT
    Q : BOOL;
    ET : TIME;
END_VAR
timeout := NONDETERMINISTIC_BOOL();
IF NOT IN THEN
    Q := FALSE;
    running := FALSE;
ELSIF NOT running AND NOT Q THEN
    running := TRUE;
ELSIF running AND NOT Q THEN
    Q := timeout;
    running := NOT Q;
END_IF;
ET := NONDETERMINISTIC_TIME();
END_FUNCTION_BLOCK

FUNCTION_BLOCK RTRIG
VAR_INPUT
    CLK : BOOL;
END_VAR
VAR
    M : BOOL;
END_VAR
VAR_OUTPUT
    Q : BOOL;
END_VAR
    Q := CLK AND NOT M;
    M := CLK;
END_FUNCTION_BLOCK

FUNCTION_BLOCK FTRIG
VAR_INPUT
    CLK : BOOL;
END_VAR
VAR
   M : BOOL;
END_VAR
VAR_OUTPUT
   Q : BOOL;
END_VAR
    Q := NOT CLK AND M;
    M := CLK;
END_FUNCTION_BLOCK

(* ---- 4.3.Muting.st ---- *)
PROGRAM Muting
VAR_INPUT
    S1SEStopIn : SAFEBOOL;
    S2MutingSwitch11 : BOOL;
    S3MutingSwitch12 : BOOL;
    S4MutingSwitch21 : BOOL;
    S5MutingSwitch22 : BOOL;
    S6SGuardSwitch : SAFEBOOL;
    L1SMutingLamp : SAFEBOOL;
    S7SAOPDIn : SAFEBOOL;
    K1SEDM : SAFEBOOL;
    K2SEDM : SAFEBOOL;
    S9Reset : BOOL;
    S0Reset : BOOL;
    ApplCtrl1 : BOOL;
    StartTestLC1 : BOOL;
    ApplMutingEnable1 : BOOL;
END_VAR
VAR
    SSafeControl : SAFEBOOL := TRUE;
    SFEmergencyStop1 : SFEmergencyStop;
    SFGuardMonitoring1 : SFGuardMonitoring;
    SFMutingSeq1 : SFMutingSeq;
    SFLightCurtain1 : SFTestableSafetySensor;
    SFOutControl1 : SFOutControl;
    SFEDM1 : SFEDM;
END_VAR
VAR_OUTPUT
    SEDMOutK : SAFEBOOL;
    SMutingActiveL1 : SAFEBOOL;
    STestOutLightCurtainS8 : SAFEBOOL;
    ErrorEStop1 : BOOL;
    DiagEStop1 : WORD;
    ErrorGuard1 : BOOL;
    DiagGuard1 : WORD;
    ErrorMuting1 : BOOL;
    DiagMuting1 : WORD;
    ErrorLightCurtain1 : BOOL;
    DiagLightCurtain1 : WORD;
    ErrorOutControl1 : BOOL;
    DiagOutControl1 : WORD;
    ErrorEDM1 : BOOL;
    DiagEDM1 : WORD;
    TestPossibleLC1 : BOOL;
    TestExecutedLC1 : BOOL;
END_VAR
SFEmergencyStop1(Activate:=TRUE, SEStopIn:=S1SEStopIn, SStartReset:=TRUE, SAutoReset:=FALSE, Reset:=S9Reset);
ErrorEStop1 := SFEmergencyStop1.Error;
DiagEStop1 := SFEmergencyStop1.DiagCode;

SFGuardMonitoring1(Activate:=TRUE, SGuardSwitch1:=S6SGuardSwitch, SGuardSwitch2:=S6SGuardSwitch, DiscrepancyTime:=T#0ms, SStartReset:=TRUE, SAutoReset:=FALSE, Reset:=S9Reset);
ErrorGuard1 := SFGuardMonitoring1.Error;
DiagGuard1 := SFGuardMonitoring1.DiagCode;

SFLightCurtain1(Activate:=TRUE, SOSSDIn:=S7SAOPDIn, StartTest:=StartTestLC1, TestTime:=T#100ms, NoExternalTest:=TRUE, SStartReset:=TRUE, SAutoReset:=FALSE, Reset:=S0Reset);
SFMutingSeq1(Activate:=TRUE, SAOPDIn:=SFLightCurtain1.SOSSDOut, MutingSwitch11:=S2MutingSwitch11, MutingSwitch12:=S3MutingSwitch12, MutingSwitch21:=S4MutingSwitch21, MutingSwitch22:=S5MutingSwitch22,
SMutingLamp:=L1SMutingLamp, MaxMutingTime:=T#30s, MutingEnable:=ApplMutingEnable1, SStartReset:=TRUE, Reset:=S9Reset);
STestOutLightCurtainS8 := SFLightCurtain1.STestOut;
TestPossibleLC1 := SFLightCurtain1.TestPossible;
TestExecutedLC1 := SFLightCurtain1.TestExecuted;
ErrorLightCurtain1 := SFLightCurtain1.Error;
DiagLightCurtain1 := SFLightCurtain1.DiagCode;
SMutingActiveL1 := SFMutingSeq1.SMutingActive;
ErrorMuting1 := SFMutingSeq1.Error;
DiagMuting1 := SFMutingSeq1.DiagCode;

SSafeControl := SFEmergencyStop1.SEStopOut AND SFGuardMonitoring1.SGuardMonitoring AND SFMutingSeq1.SAOPDOut;

SFOutControl1(Activate:=TRUE, SSafeControl:=SSafeControl, ProcessControl:=ApplCtrl1, StaticControl:=FALSE, SStartReset:=FALSE, SAutoReset:=FALSE, Reset:=S0Reset);
ErrorOutControl1 := SFOutControl1.Error;
DiagOutControl1 := SFOutControl1.DiagCode;

SFEDM1(Activate:=TRUE, SOutControl:=SFOutControl1.SOutControl, SEDM1:=K1SEDM, SEDM2:=K2SEDM, MonitoringTime:=T#30ms, SStartReset:=FALSE, Reset:=S0Reset);
SEDMOutK := SFEDM1.SEDMOut;
ErrorEDM1 := SFEDM1.Error;
DiagEDM1 := SFEDM1.DiagCode;
END_PROGRAM

FUNCTION_BLOCK SFEmergencyStop
VAR_INPUT
    Activate : BOOL;
    SEStopIn : BOOL;
    SStartReset : BOOL;
    SAutoReset : BOOL;
    Reset : BOOL;
END_VAR
VAR
    RTRIGatReset : RTRIG;
END_VAR
VAR_OUTPUT
    Ready : BOOL;
    SEStopOut : BOOL;
    Error : BOOL;
    DiagCode : WORD;
END_VAR
RTRIGatReset(CLK:=Reset);
IF NOT Activate THEN
    DiagCode := 16#0000;
ELSE
    CASE DiagCode OF
    16#0000:
        IF Activate THEN
            DiagCode := 16#8001;
        END_IF;
    16#8001:
        IF NOT SStartReset THEN
            DiagCode := 16#8002;
        ELSIF SStartReset AND NOT SEStopIn THEN
            DiagCode := 16#8004;
        ELSIF SEStopIn AND SStartReset THEN
            DiagCode := 16#8000;
        END_IF;
    16#8002:
        IF SEStopIn THEN
            DiagCode := 16#8003;
        END_IF;
    16#8003:
        IF Reset AND NOT RTRIGatReset.Q THEN
            DiagCode := 16#C001;
        ELSIF NOT SEStopIn THEN
            DiagCode := 16#8002;
        ELSIF RTRIGatReset.Q THEN
            DiagCode := 16#8000;
        END_IF;
    16#C001:
        IF NOT Reset THEN
            DiagCode := 16#8003;
        END_IF;
    16#8004:
        IF SEStopIn AND NOT SAutoReset THEN
            DiagCode := 16#8005;
        ELSIF SEStopIn AND SAutoReset THEN
            DiagCode := 16#8000;
        END_IF;
    16#8005:
        IF Reset AND NOT RTRIGatReset.Q THEN
            DiagCode := 16#C002;
        ELSIF NOT SEStopIn THEN
            DiagCode := 16#8004;
        ELSIF RTRIGatReset.Q OR SAutoReset THEN
            DiagCode := 16#8000;
        END_IF;
    16#C002:
        IF NOT Reset THEN
            DiagCode := 16#8005;
        END_IF;
    16#8000:
        IF NOT SEStopIn THEN
            DiagCode := 16#8004;
        END_IF;
    END_CASE;
END_IF;
CASE DiagCode OF
16#0000:
    Ready := FALSE;
    Error := FALSE;
    SEStopOut := FALSE;
16#8001:
    Ready := TRUE;
    Error := FALSE;
    SEStopOut := FALSE;
16#8002:
    Ready := TRUE;
    Error := FALSE;
    SEStopOut := FALSE;
16#8003:
    Ready := TRUE;
    Error := FALSE;
    SEStopOut := FALSE;
16#C001:
    Ready := TRUE;
    Error := TRUE;
    SEStopOut := FALSE;
16#8004:
    Ready := TRUE;
    Error := FALSE;
    SEStopOut := FALSE;
16#8005:
    Ready := TRUE;
    Error := FALSE;
    SEStopOut := FALSE;
16#C002:
    Ready := TRUE;
    Error := TRUE;
    SEStopOut := FALSE;
16#8000:
    Ready := TRUE;
    Error := FALSE;
    SEStopOut := TRUE;
END_CASE;
END_FUNCTION_BLOCK

FUNCTION_BLOCK SFGuardMonitoring
VAR_INPUT
    Activate : BOOL := FALSE;
    SGuardSwitch1 : SAFEBOOL := FALSE;
    SGuardSwitch2 : SAFEBOOL := FALSE;
    DiscrepancyTime : TIME := T#0s;
    SStartReset : SAFEBOOL := FALSE;
    SAutoReset : SAFEBOOL := FALSE;
    Reset : BOOL := FALSE;
END_VAR
VAR
    Timer : TON;
    RTRIGatReset : RTRIG;
END_VAR
VAR_OUTPUT
    Ready : BOOL := FALSE;
    SGuardMonitoring : BOOL := FALSE;
    Error : BOOL := FALSE;
    DiagCode : WORD := 16#0000;
END_VAR
RTRIGatReset(CLK:=Reset);
IF NOT Activate THEN
    DiagCode := 16#0000;
ELSE
    CASE DiagCode OF
    16#0000:
        IF Activate THEN
            DiagCode := 16#8001;
        END_IF;
    16#8001:
        IF NOT SGuardSwitch1 OR NOT SGuardSwitch2 THEN
            DiagCode := 16#8002;
        ELSIF SGuardSwitch1 AND SGuardSwitch2 AND NOT SStartReset THEN
            DiagCode := 16#8003;
        ELSIF SGuardSwitch1 AND SGuardSwitch2 AND SStartReset THEN
            DiagCode := 16#8000;
        END_IF;
    16#8002:
        IF NOT SGuardSwitch1 AND NOT SGuardSwitch2 THEN
            DiagCode := 16#8012;
        END_IF;
    16#8003:
        IF Reset AND NOT RTRIGatReset.Q THEN
            DiagCode := 16#C001;
        ELSIF NOT SGuardSwitch1 OR NOT SGuardSwitch2 THEN
            DiagCode := 16#8002;
        ELSIF RTRIGatReset.Q THEN
            DiagCode := 16#8000;
        END_IF;
    16#8012:
        IF SGuardSwitch1 THEN
            DiagCode := 16#8004;
        ELSIF SGuardSwitch2 THEN
            DiagCode := 16#8014;
        END_IF;
    16#8004:
        IF Timer.Q THEN
            DiagCode := 16#C011;
        ELSIF NOT SGuardSwitch1 THEN
            DiagCode := 16#8002;
        ELSIF SGuardSwitch2 THEN
            DiagCode := 16#8005;
        END_IF;
    16#8014:
        IF Timer.Q THEN
            DiagCode := 16#C012;
        ELSIF NOT SGuardSwitch2 THEN
            DiagCode := 16#8002;
        ELSIF SGuardSwitch1 THEN
            DiagCode := 16#8005;
        END_IF;
    16#8005:
        IF NOT SGuardSwitch1 OR NOT SGuardSwitch2 THEN
            DiagCode := 16#8002;
        ELSIF NOT SAutoReset THEN
            DiagCode := 16#8003;
        ELSIF SAutoReset THEN
            DiagCode := 16#8000;
        END_IF;
    16#8000:
        IF NOT SGuardSwitch1 OR NOT SGuardSwitch2 THEN
            DiagCode := 16#8002;
        END_IF;
    16#C001:
        IF NOT Reset THEN
            DiagCode := 16#8003;
        END_IF;
    16#C011:
        IF NOT SGuardSwitch1 AND NOT SGuardSwitch2 THEN
            DiagCode := 16#8012;
        END_IF;
    16#C012:
        IF NOT SGuardSwitch1 AND NOT SGuardSwitch2 THEN
            DiagCode := 16#8012;
        END_IF;
    END_CASE;
END_IF;
CASE DiagCode OF
16#0000:
    Timer(IN:=FALSE, PT:=DiscrepancyTime);
    Ready := FALSE;
    Error := FALSE;
    SGuardMonitoring := FALSE;
16#8000:
    Timer(IN:=FALSE, PT:=DiscrepancyTime);
    Ready := TRUE;
    Error := FALSE;
    SGuardMonitoring  := TRUE;
16#8001,
16#8002,
16#8003,
16#8012,
16#8005:
    Timer(IN:=FALSE, PT:=DiscrepancyTime);
    Ready := TRUE;
    Error := FALSE;
    SGuardMonitoring := FALSE;
16#8004,
16#8014:
    Timer(IN:=TRUE, PT:=DiscrepancyTime);
    Ready := TRUE;
    Error := FALSE;
    SGuardMonitoring := FALSE;
16#C001,
16#C011,
16#C012:
    Timer(IN:=FALSE, PT:=DiscrepancyTime);
    Ready := TRUE;
    Error := TRUE;
    SGuardMonitoring := FALSE;
END_CASE;
END_FUNCTION_BLOCK

FUNCTION_BLOCK SFMutingSeq
VAR_INPUT
    Activate : BOOL := FALSE;
    SAOPDIn : SAFEBOOL := FALSE;
    MutingSwitch11 : BOOL := FALSE;
    MutingSwitch12 : BOOL := FALSE;
    MutingSwitch21 : BOOL := FALSE;
    MutingSwitch22 : BOOL := FALSE;
    SMutingLamp : SAFEBOOL := FALSE;
    DiscTime1112 : TIME := T#0s;
    DiscTime2122 : TIME := T#0s;
    MaxMutingTime : TIME := T#0s;
    MutingEnable : BOOL := FALSE;
    SStartReset : SAFEBOOL := FALSE;
    Reset : BOOL := FALSE;
END_VAR
VAR
    Timer : TON;
    RTRIGatReset : RTRIG;
    RTRIGatMS11 : RTRIG;
    RTRIGatMS12 : RTRIG;
    RTRIGatMS21 : RTRIG;
    RTRIGatMS22 : RTRIG;
    FTRIGatMS11 : FTRIG;
    FTRIGatMS12 : FTRIG;
    FTRIGatMS21 : FTRIG;
    FTRIGatMS22 : FTRIG;
END_VAR
VAR_OUTPUT
    Ready : BOOL := FALSE;
    SAOPDOut : SAFEBOOL := FALSE;
    SMutingActive : SAFEBOOL := FALSE;
    Error : BOOL := FALSE;
    DiagCode : WORD := 16#0000;
END_VAR
RTRIGatReset(CLK:=Reset);
RTRIGatMS11(CLK:=MutingSwitch11);
RTRIGatMS12(CLK:=MutingSwitch12);
RTRIGatMS21(CLK:=MutingSwitch21);
RTRIGatMS22(CLK:=MutingSwitch22);
FTRIGatMS11(CLK:=MutingSwitch11);
FTRIGatMS12(CLK:=MutingSwitch12);
FTRIGatMS21(CLK:=MutingSwitch21);
FTRIGatMS22(CLK:=MutingSwitch22);
IF NOT Activate THEN
    DiagCode := 16#0000;
ELSE
    CASE DiagCode OF
    16#0000:
    IF Activate THEN
        DiagCode := 16#8001;
    END_IF;
    16#8000:
        IF (NOT MutingEnable AND RTRIGatMS11.Q) OR (NOT MutingEnable AND RTRIGatMS22.Q) OR (MutingSwitch12 OR MutingSwitch21) OR (MutingSwitch11 AND MutingSwitch22) THEN
            (* Wrong muting sequence *)
            DiagCode := 16#C004;
        ELSIF NOT SAOPDIn THEN
            DiagCode := 16#8002;
        ELSIF NOT SMutingLamp THEN
            DiagCode := 16#C003;
        ELSIF MutingEnable AND (RTRIGatMS11.Q AND NOT MutingSwitch12 AND NOT MutingSwitch21 AND NOT MutingSwitch22) THEN
            DiagCode := 16#8011;
            Timer(IN:=TRUE, PT:=MaxMutingTime);
        ELSIF MutingEnable AND (NOT MutingSwitch11 AND NOT MutingSwitch12 AND NOT MutingSwitch21 AND RTRIGatMS22.Q) THEN
            DiagCode := 16#8122;
            Timer(IN:=TRUE, PT:=MaxMutingTime);
        END_IF;
    16#8001:
        IF Reset AND NOT RTRIGatReset.Q AND NOT SStartReset THEN
            DiagCode := 16#C001;
        (*
        ELSIF (Time parameters out of range)
        DiagCode := 16#C005;
        *)
        ELSIF RTRIGatReset.Q OR SStartReset THEN
            DiagCode := 16#8005;
        END_IF;
    16#8002:
        IF SAOPDIn THEN
            DiagCode := 16#8003;
        END_IF;
    16#8003:
        IF Reset AND NOT RTRIGatReset.Q THEN
            DiagCode := 16#C002;
        ELSIF RTRIGatReset.Q THEN
            DiagCode := 16#8005;
        END_IF;
    16#8005:
        IF NOT SAOPDIn THEN
            DiagCode := 16#8002;
        ELSIF NOT SMutingLamp THEN
            DiagCode := 16#C003;
        ELSIF SAOPDIn THEN
            DiagCode := 16#8000;
        END_IF;
    16#C001:
        IF NOT Reset THEN
            DiagCode := 16#8001;
        END_IF;
    16#C002:
        IF NOT Reset THEN
            DiagCode := 16#8003;
        END_IF;
    16#C003:
        IF SMutingLamp THEN
            DiagCode := 16#8003;
        END_IF;
    16#C006,
    16#C007,
    16#C008:
        IF NOT (MutingSwitch11 OR MutingSwitch12 OR MutingSwitch21 OR MutingSwitch22) THEN
            DiagCode := 16#8003;
        END_IF;
    ELSE
        IF DiagCode >= 16#C000 THEN
        (* 16#CYx4 *)
            IF NOT (MutingSwitch11 OR MutingSwitch12 OR MutingSwitch21 OR MutingSwitch22) THEN
                DiagCode := 16#8003;
            END_IF;
        ELSE
            (* cases 16#8011 .. 16#8422 *)
            CASE DiagCode OF
            16#8011:
                IF NOT MutingEnable OR NOT MutingSwitch11 OR MutingSwitch21 OR MutingSwitch22 THEN
                    DiagCode := 16#C104;
                ELSIF Timer.Q THEN
                    DiagCode := 16#C006;
                ELSIF NOT SAOPDIn THEN
                    DiagCode := 16#8002;
                ELSIF NOT SMutingLamp THEN
                    DiagCode := 16#C003;
                ELSIF MutingEnable AND (MutingSwitch11 AND RTRIGatMS12.Q AND NOT MutingSwitch21 AND NOT MutingSwitch22) THEN
                    DiagCode := 16#8012;
                END_IF;
            16#8012:
                IF RTRIGatMS11.Q OR RTRIGatMS12.Q OR FTRIGatMS22.Q THEN
                    DiagCode := 16#C104;
                ELSIF Timer.Q THEN
                    DiagCode := 16#C006;
                ELSIF NOT SMutingLamp THEN
                    DiagCode := 16#C003;
                ELSIF NOT MutingSwitch11 AND NOT MutingSwitch12 AND FTRIGatMS21.Q AND MutingSwitch22 THEN
                    Timer(IN:=FALSE, PT:=MaxMutingTime);
                    DiagCode := 16#8000;
                END_IF;
            16#8122:
                IF NOT MutingEnable OR MutingSwitch11 OR MutingSwitch12 OR NOT MutingSwitch22 THEN
                    DiagCode := 16#C104;
                ELSIF Timer.Q THEN
                    DiagCode := 16#C006;
                ELSIF NOT SAOPDIn THEN
                    DiagCode := 16#8002;
                ELSIF NOT SMutingLamp THEN
                    DiagCode := 16#C003;
                ELSIF MutingEnable AND (NOT MutingSwitch11 AND NOT MutingSwitch12 AND RTRIGatMS21.Q AND MutingSwitch22) THEN
                    DiagCode := 16#8112;
                END_IF;
            16#8112:
                IF FTRIGatMS11.Q OR RTRIGatMS21.Q OR RTRIGatMS22.Q THEN
                    DiagCode := 16#C104;
                ELSIF Timer.Q THEN
                    DiagCode := 16#C006;
                ELSIF NOT SMutingLamp THEN
                    DiagCode := 16#C003;
                ELSIF MutingSwitch11 AND FTRIGatMS12.Q AND NOT MutingSwitch21 AND NOT MutingSwitch22 THEN
                    DiagCode := 16#8000;
                    Timer(IN:=FALSE, PT:=MaxMutingTime);
                END_IF;
            END_CASE;
        END_IF;
    END_CASE;
END_IF;
CASE DiagCode OF
16#0000:
    Ready := FALSE;
    SAOPDOut := FALSE;
    SMutingActive := FALSE;
    Error := FALSE;
16#8000,
16#8011,
16#8122:
    Ready := TRUE;
    SAOPDOut := TRUE;
    SMutingActive := FALSE;
    Error := FALSE;
16#8001,
16#8002,
16#8003,
16#8005:
    Ready := TRUE;
    SAOPDOut := FALSE;
    SMutingActive := FALSE;
    Error := FALSE;
16#8012,
16#8112:
    Ready := TRUE;
    SAOPDOut := TRUE;
    SMutingActive := TRUE;
    Error := FALSE;
ELSE
    Ready := TRUE;
    SAOPDOut := FALSE;
    SMutingActive := FALSE;
    Error := TRUE;
END_CASE;
END_FUNCTION_BLOCK

FUNCTION_BLOCK SFTestableSafetySensor
VAR_INPUT
    Activate : BOOL;
    SOSSDIn : SAFEBOOL;
    StartTest : BOOL;
    TestTime : TIME := T#10ms;
    NoExternalTest : BOOL;
    SStartReset : SAFEBOOL;
    SAutoReset : SAFEBOOL;
    Reset : BOOL;
END_VAR
VAR
    Timer1: TON;
    Timer2: TON;
    RTRIGatReset : RTRIG;
    RTRIGatStartTest : RTRIG;
    FTRIGatSOSSDIn : FTRIG;
END_VAR
VAR_OUTPUT
    Ready : SAFEBOOL;
    SOSSDOut : SAFEBOOL;
    STestOut : SAFEBOOL := TRUE;
    TestPossible : BOOL;
    TestExecuted : BOOL;
    Error : BOOL;
    DiagCode : WORD := 16#0000;
END_VAR
RTRIGatReset(CLK:=Reset);
RTRIGatStartTest(CLK:=StartTest);
FTRIGatSOSSDIn(CLK:=SOSSDIn);
IF NOT Activate THEN
    DiagCode := 16#0000;
ELSE
    CASE DiagCode OF
    16#0000:
        IF Activate THEN
            DiagCode := 16#8001;
        END_IF;
    16#8000:
        IF NOT SOSSDIn THEN
            DiagCode := 16#8012;
        ELSIF RTRIGatStartTest.Q THEN
            DiagCode := 16#8020;
            Timer1(IN:=FALSE);
        END_IF;
    16#8001:
        IF TestTime > T#150ms THEN
            DiagCode := 16#C000;
        ELSIF Reset AND NOT RTRIGatReset.Q AND NOT SStartReset THEN
            DiagCode := 16#C001;
        ELSIF NOT SOSSDIn THEN
            DiagCode := 16#8002;
        ELSIF SOSSDIn AND (RTRIGatReset.Q OR SStartReset) THEN
            DiagCode := 16#8010;
        END_IF;
    16#8002:
        IF SOSSDIn THEN
            DiagCode := 16#8003;
        END_IF;
    16#8003:
        IF Reset AND NOT RTRIGatReset.Q AND NOT SAutoReset THEN
            DiagCode := 16#C002;
        ELSIF NOT SOSSDIn THEN
            DiagCode := 16#8002;
        ELSIF SOSSDIn AND (RTRIGatReset.Q OR SAutoReset) THEN
            DiagCode := 16#8010;
        END_IF;
    16#8004:
        IF FTRIGatSOSSDIn.Q THEN
            DiagCode := 16#8005;
        END_IF;
    16#8005:
        IF SOSSDIn THEN
            DiagCode := 16#8006;
        END_IF;
    16#8006:
        IF Reset AND NOT RTRIGatReset.Q THEN
            DiagCode := 16#C005;
        ELSIF RTRIGatReset.Q AND NOT SOSSDIn THEN
            DiagCode := 16#8002;
        ELSIF RTRIGatReset.Q AND SOSSDIn THEN
            DiagCode := 16#8010;
        END_IF;
    16#8010:
        IF NOT SOSSDIn THEN
            DiagCode := 16#8002;
        ELSIF RTRIGatStartTest.Q THEN
            DiagCode := 16#8020;
            Timer1(IN:=FALSE);
        END_IF;
    16#8012:
        IF SOSSDIn THEN
            DiagCode := 16#8013;
        END_IF;
    16#8013:
        IF Reset AND NOT RTRIGatReset.Q AND NOT SAutoReset THEN
            DiagCode := 16#C007;
        ELSIF NOT SOSSDIn THEN
            DiagCode := 16#8012;
        ELSIF SOSSDIn AND (RTRIGatReset.Q OR SAutoReset) THEN
            DiagCode := 16#8000;
        END_IF;
    16#8020:
        IF Timer1.Q THEN
            DiagCode := 16#C020;
        ELSIF NOT SOSSDIn THEN
            DiagCode := 16#8030;
            Timer2(IN:=FALSE);
        END_IF;
    16#8030:
        IF Timer2.Q THEN
            DiagCode := 16#C030;
        ELSIF SOSSDIn THEN
            DiagCode := 16#8000;
        END_IF;
    16#C000:
        IF Reset AND NOT RTRIGatReset.Q THEN
            DiagCode := 16#C006;
        ELSIF RTRIGatReset.Q AND TestTime <= T#150ms THEN
            DiagCode := 16#8001;
        END_IF;
    16#C001:
        IF NOT Reset THEN
            DiagCode := 16#8001;
        END_IF;
    16#C002:
        IF NOT Reset THEN
            DiagCode := 16#8003;
        END_IF;
    16#C003:
        IF NOT Reset THEN
            DiagCode := 16#C010;
        END_IF;
    16#C004:
        IF NOT Reset THEN
            DiagCode := 16#C020;
        END_IF;
    16#C005:
        IF NOT Reset THEN
            DiagCode := 16#8006;
        END_IF;
    16#C006:
        IF NOT Reset THEN
            DiagCode := 16#C000;
        END_IF;
    16#C007:
        IF NOT Reset THEN
            DiagCode := 16#8013;
        END_IF;
    16#C010:
        IF Reset AND NOT RTRIGatReset.Q THEN
            DiagCode := 16#C003;
        ELSIF RTRIGatReset.Q AND NOT NoExternalTest THEN
            DiagCode := 16#8004;
        ELSIF SOSSDIn AND (RTRIGatReset.Q AND NoExternalTest) THEN
            DiagCode := 16#8010;
        END_IF;
    16#C020:
        IF Reset AND NOT RTRIGatReset.Q THEN
            DiagCode := 16#C004;
        ELSIF RTRIGatReset.Q AND NOT NoExternalTest THEN
            DiagCode := 16#8004;
        ELSIF SOSSDIn AND (RTRIGatReset.Q AND NoExternalTest) THEN
            DiagCode := 16#8010;
        END_IF;
    END_CASE;
END_IF;
CASE DiagCode OF
16#0000:
    Ready := FALSE;
    SOSSDOut := FALSE;
    STestOut := TRUE;
    TestPossible := FALSE;
    TestExecuted := FALSE;
    Error := FALSE;
16#8000:
    Ready := TRUE;
    SOSSDOut := TRUE;
    STestOut := TRUE;
    TestPossible := TRUE;
    TestExecuted := TRUE;
    Error := FALSE;
16#8001, 16#8002, 16#8003, 16#8004, 16#8005, 16#8006:
    Ready := TRUE;
    SOSSDOut := FALSE;
    STestOut := TRUE;
    TestPossible := FALSE;
    TestExecuted := FALSE;
    Error := FALSE;
16#8010:
    Ready := TRUE;
    SOSSDOut := TRUE;
    STestOut := TRUE;
    TestPossible := TRUE;
    TestExecuted := FALSE;
    Error := FALSE;
16#8012, 16#8013:
    Ready := TRUE;
    SOSSDOut := FALSE;
    STestOut := TRUE;
    TestPossible := FALSE;
    TestExecuted := TRUE;
    Error := FALSE;
16#8020:
    Ready := TRUE;
    SOSSDOut := TRUE;
    STestOut := FALSE;
    TestPossible := FALSE;
    TestExecuted := FALSE;
    Error := FALSE;
    Timer1(IN:=TRUE, PT:=TestTime);
16#8030:
    Ready := TRUE;
    SOSSDOut := TRUE;
    STestOut := TRUE;
    TestPossible := FALSE;
    TestExecuted := FALSE;
    Error := FALSE;
    Timer2(IN:=TRUE, PT:=TestTime);
16#C000, 16#C001, 16#C002, 16#C003, 16#C004, 16#C005, 16#C006, 16#C010, 16#C020:
    Ready := TRUE;
    SOSSDOut := FALSE;
    STestOut := TRUE;
    TestPossible := FALSE;
    TestExecuted := FALSE;
    Error := TRUE;
16#C007:
    Ready := TRUE;
    SOSSDOut := FALSE;
    STestOut := TRUE;
    TestPossible := FALSE;
    TestExecuted := TRUE;
    Error := TRUE;
END_CASE;
END_FUNCTION_BLOCK

FUNCTION_BLOCK SFOutControl
VAR_INPUT
    Activate : BOOL ;
    SSafeControl : SAFEBOOL ;
    ProcessControl : BOOL ;
    StaticControl : BOOL ;
    SStartReset : SAFEBOOL ;
    SAutoReset	: SAFEBOOL ;
    Reset : BOOL ;
END_VAR
VAR
    RTRIGatReset : RTRIG ;
    RTRIGatProcessControl : RTRIG ;
END_VAR
VAR_OUTPUT
    Ready : BOOL ;
    SOutControl : SAFEBOOL ;
    Error : BOOL ;
    DiagCode : WORD:=16#0000 ;
END_VAR
RTRIGatReset(CLK:=Reset);
RTRIGatProcessControl(CLK:=ProcessControl);
IF NOT Activate THEN
    DiagCode := 16#0000;
ELSE
    CASE DiagCode OF
    16#0000:
        IF Activate THEN
            DiagCode := 16#8001;
        END_IF;
    16#8000:
        IF NOT SSafeControl THEN
            DiagCode := 16#8002;
        ELSIF NOT ProcessControl THEN
            DiagCode := 16#8010;
        END_IF;
    16#8001:
        IF Reset AND NOT RTRIGatReset.Q AND NOT SStartReset THEN
            DiagCode := 16#C001;
        ELSIF RTRIGatReset.Q AND RTRIGatProcessControl.Q THEN
            DiagCode := 16#C111;
        ELSIF RTRIGatReset.Q OR SStartReset THEN
            DiagCode := 16#8010;
        END_IF;
    16#8002:
        IF SSafeControl THEN
            DiagCode := 16#8003;
        END_IF;
    16#8003:
        IF NOT SSafeControl THEN
            DiagCode := 16#8002;
        ELSIF Reset AND NOT RTRIGatReset.Q AND NOT SAutoReset THEN
            DiagCode := 16#C002;
        ELSIF RTRIGatReset.Q AND RTRIGatProcessControl.Q THEN
            DiagCode := 16#C211;
        ELSIF RTRIGatReset.Q OR SAutoReset THEN
            DiagCode := 16#8010;
        END_IF;
    16#8010:
        IF NOT SSafeControl THEN
            DiagCode := 16#8002;
        ELSIF NOT RTRIGatProcessControl.Q AND ProcessControl AND NOT StaticControl THEN
            DiagCode := 16#C010;
        ELSIF SSafeControl AND (RTRIGatProcessControl.Q OR (StaticControl AND ProcessControl)) THEN
            DiagCode := 16#8000;
        END_IF;
    16#C001:
        IF NOT Reset THEN
            DiagCode := 16#8001;
        END_IF;
    16#C002:
        IF NOT Reset THEN
            DiagCode := 16#8003;
        END_IF;
    16#C010:
        IF NOT ProcessControl THEN
            DiagCode := 16#8010;
        END_IF;
    16#C111:
        IF NOT Reset THEN
            DiagCode := 16#8001;
        END_IF;
    16#C211:
        IF NOT Reset THEN
            DiagCode := 16#8003;
        END_IF;
    END_CASE;
END_IF;
CASE DiagCode OF
16#0000:
    Ready := FALSE;
    SOutControl := FALSE;
    Error := FALSE;
16#8000:
    Ready := TRUE;
    SOutControl := TRUE;
    Error := FALSE;
16#8001, 16#8002, 16#8003, 16#8010:
    Ready := TRUE;
    SOutControl := FALSE;
    Error := FALSE;
16#C001, 16#C002, 16#C010, 16#C111, 16#C211:
    Ready := TRUE;
    SOutControl := FALSE;
    Error := TRUE;
END_CASE;
END_FUNCTION_BLOCK

FUNCTION_BLOCK SFEDM
VAR_INPUT
    Activate : BOOL ;
    SOutControl	: SAFEBOOL ;
    SEDM1 : SAFEBOOL ;
    SEDM2 : SAFEBOOL ;
    MonitoringTime : TIME;
    SStartReset	: SAFEBOOL ;
    Reset : BOOL ;
END_VAR
VAR
    Timer : TON;
    RTRIGatReset : RTRIG ;
    RTRIGatOutControl : RTRIG ;
    RTRIGatEDM1 : RTRIG ;
    RTRIGatEDM2	: RTRIG ;
END_VAR
VAR_OUTPUT
    Ready : BOOL ;
    SEDMOut	: SAFEBOOL ;
    Error : BOOL ;
    DiagCode : WORD:=16#0000 ;
END_VAR
(* Rising edge detection *)
RTRIGatReset(CLK:=Reset);
RTRIGatOutControl(CLK:=SOutControl);
RTRIGatEDM1(CLK:=SEDM1);
RTRIGatEDM2(CLK:=SEDM2);
IF NOT Activate THEN
    DiagCode := 16#0000;
ELSE
    CASE DiagCode OF
    16#0000:
        IF Activate THEN
            DiagCode := 16#8001;
        END_IF;
    16#8000:
        IF Timer.Q AND SEDM1 AND NOT SEDM2 THEN
            DiagCode := 16#C070;
        ELSIF Timer.Q AND NOT SEDM1 AND SEDM2 THEN
            DiagCode := 16#C080;
        ELSIF Timer.Q AND SEDM1 AND SEDM2 THEN
            DiagCode := 16#C090;
        ELSIF NOT SOutControl THEN
            DiagCode := 16#8010;
            Timer(IN:=FALSE);
        END_IF;
    16#8001:
        IF Reset AND NOT RTRIGatReset.Q AND NOT SStartReset THEN
            DiagCode := 16#C001;
        ELSIF RTRIGatReset.Q AND RTRIGatOutControl.Q AND NOT SStartReset THEN
            DiagCode := 16#C111;
        ELSIF RTRIGatReset.Q OR SStartReset THEN
            DiagCode := 16#8010;
            Timer(IN:=FALSE);
        END_IF;
    16#8010:
        IF SOutControl AND NOT SEDM1 AND SEDM2 THEN
            DiagCode := 16#C010;
        ELSIF SOutControl AND SEDM1 AND NOT SEDM2 THEN
            DiagCode := 16#C020;
        ELSIF SOutControl AND NOT SEDM1 AND NOT SEDM2 THEN
            DiagCode := 16#C030;
        ELSIF Timer.Q AND NOT SEDM1 AND SEDM2 THEN
            DiagCode := 16#C040;
        ELSIF Timer.Q AND SEDM1 AND NOT SEDM2 THEN
            DiagCode := 16#C050;
        ELSIF Timer.Q AND NOT SEDM1 AND NOT SEDM2 THEN
            DiagCode := 16#C060;
        ELSIF SOutControl THEN
            DiagCode := 16#8000;
            Timer(IN:=FALSE);
        END_IF;
    16#C001:
        IF NOT Reset THEN
            DiagCode := 16#8001;
        END_IF;
    16#C010, 16#C020, 16#C030:
        IF (Reset AND NOT RTRIGatReset.Q AND SEDM1 AND SEDM2) OR (RTRIGatReset.Q AND RTRIGatEDM1.Q AND NOT RTRIGatEDM2.Q) THEN
            DiagCode := 16#C011;
        ELSIF (Reset AND NOT RTRIGatReset.Q AND SEDM1 AND SEDM2) OR (RTRIGatReset.Q AND NOT RTRIGatEDM1.Q AND RTRIGatEDM2.Q) THEN
            DiagCode := 16#C021;
        ELSIF (Reset AND NOT RTRIGatReset.Q AND SEDM1 AND SEDM2) OR (RTRIGatReset.Q AND RTRIGatEDM1.Q AND RTRIGatEDM2.Q) THEN
            DiagCode := 16#C031;
        ELSIF RTRIGatReset.Q AND SEDM1 AND SEDM2 THEN
            DiagCode := 16#8010;
            Timer(IN:=FALSE);
        END_IF;
    16#C011:
        IF NOT Reset THEN
            DiagCode := 16#C010;
        END_IF;
    16#C021:
        IF NOT Reset THEN
            DiagCode := 16#C020;
        END_IF;
    16#C031:
        IF NOT Reset THEN
            DiagCode := 16#C030;
        END_IF;
    16#C040, 16#C050, 16#C060:
        IF (Reset AND NOT RTRIGatReset.Q AND SEDM1 AND SEDM2) OR (RTRIGatReset.Q AND RTRIGatEDM1.Q AND NOT RTRIGatEDM2.Q) THEN
            DiagCode := 16#C041;
        ELSIF (Reset AND NOT RTRIGatReset.Q AND SEDM1 AND SEDM2) OR (RTRIGatReset.Q AND NOT RTRIGatEDM1.Q AND RTRIGatEDM2.Q) THEN
            DiagCode := 16#C051;
        ELSIF (Reset AND NOT RTRIGatReset.Q AND SEDM1 AND SEDM2) OR (RTRIGatReset.Q AND RTRIGatEDM1.Q AND RTRIGatEDM2.Q) THEN
            DiagCode := 16#C061;
        ELSIF RTRIGatReset.Q AND SEDM1 AND SEDM2 THEN
            DiagCode := 16#8010;
            Timer(IN:=FALSE);
        END_IF;
    16#C041:
        IF NOT Reset THEN
            DiagCode := 16#C040;
        END_IF;
    16#C051:
        IF NOT Reset THEN
            DiagCode := 16#C050;
        END_IF;
    16#C061:
        IF NOT Reset THEN
            DiagCode := 16#C060;
        END_IF;
    16#C070:
        IF Reset AND NOT RTRIGatReset.Q THEN
            DiagCode := 16#C071;
        ELSIF RTRIGatReset.Q AND NOT (RTRIGatEDM1.Q OR RTRIGatEDM2.Q) THEN
            DiagCode := 16#8010;
            Timer(IN:=FALSE);
        END_IF;
    16#C080:
        IF Reset AND NOT RTRIGatReset.Q THEN
            DiagCode := 16#C081;
        ELSIF RTRIGatReset.Q AND NOT (RTRIGatEDM1.Q OR RTRIGatEDM2.Q) THEN
            DiagCode := 16#8010;
            Timer(IN:=FALSE);
        END_IF;
    16#C090:
        IF Reset AND NOT RTRIGatReset.Q THEN
            DiagCode := 16#C091;
        ELSIF RTRIGatReset.Q AND NOT (RTRIGatEDM1.Q OR RTRIGatEDM2.Q) THEN
            DiagCode := 16#8010;
            Timer(IN:=FALSE);
        END_IF;
    16#C071:
        IF NOT Reset THEN
            DiagCode := 16#C070;
        END_IF;
    16#C081:
        IF NOT Reset THEN
            DiagCode := 16#C080;
        END_IF;
    16#C091:
        IF NOT Reset THEN
            DiagCode := 16#C090;
        END_IF;
    16#C111:
        IF NOT Reset THEN
            DiagCode := 16#8001;
        END_IF;
    END_CASE;
END_IF;
CASE DiagCode OF
16#0000:
    Ready := FALSE;
    SEDMOut := FALSE;
    Error := FALSE;
16#8001:
    Ready := TRUE;
    SEDMOut := FALSE;
    Error := FALSE;
16#8010:
    Ready := TRUE;
    SEDMOut := FALSE;
    Error := FALSE;
    Timer(IN:=TRUE, PT:=MonitoringTime);
16#8000:
    Ready := TRUE;
    SEDMOut := TRUE;
    Error := FALSE;
    Timer(IN:=TRUE, PT:=MonitoringTime);
16#C001, 16#C010, 16#C011, 16#C020, 16#C021, 16#C030, 16#C031, 16#C040, 16#C041, 16#C050, 16#C051, 16#C060, 16#C061, 16#C070, 16#C071, 16#C080, 16#C081, 16#C090, 16#C091, 16#C111:
    Ready := TRUE;
    SEDMOut := FALSE;
    Error := TRUE;
END_CASE;
END_FUNCTION_BLOCK

FUNCTION_BLOCK TON
VAR_INPUT
    IN : BOOL;
    PT : TIME;
END_VAR
VAR
    running : BOOL;
END_VAR
VAR_TEMP
    timeout : BOOL;
END_VAR
VAR_OUTPUT
    Q : BOOL;
    ET : TIME;
END_VAR
timeout := NONDETERMINISTIC_BOOL();
IF NOT IN THEN
    Q := FALSE;
    running := FALSE;
ELSIF NOT running AND NOT Q THEN
    running := TRUE;
ELSIF running AND NOT Q THEN
    Q := timeout;
    running := NOT Q;
END_IF;
ET := NONDETERMINISTIC_TIME();
END_FUNCTION_BLOCK

FUNCTION_BLOCK RTRIG
VAR_INPUT
    CLK : BOOL;
END_VAR
VAR
    M : BOOL;
END_VAR
VAR_OUTPUT
    Q : BOOL;
END_VAR
    Q := CLK AND NOT M;
    M := CLK;
END_FUNCTION_BLOCK

FUNCTION_BLOCK FTRIG
VAR_INPUT
    CLK : BOOL;
END_VAR
VAR
   M : BOOL;
END_VAR
VAR_OUTPUT
   Q : BOOL;
END_VAR
    Q := NOT CLK AND M;
    M := CLK;
END_FUNCTION_BLOCK

(* ---- 4.4.SafeMotionIO.st ---- *)
PROGRAM SafeMotionIO
VAR_INPUT
    S1SEStopIn : SAFEBOOL;
    S2SAutoMode : SAFEBOOL;
    S2SSetupMode : SAFEBOOL;
    S4SEnableSwitchCh1 : SAFEBOOL;
    S4SEnableSwitchCh2 : SAFEBOOL;
    S5SGuardSwitch : SAFEBOOL;
    S7SGuardLock : SAFEBOOL;
    S0Reset : BOOL;
    S8UnlockGuard : BOOL;
    M1SAcknowledgeSS1 : SAFEBOOL;
    M1SAcknowledgeSafeMotion : SAFEBOOL;
END_VAR
VAR
    SSetupMode : SAFEBOOL;
    SAutoMode : SAFEBOOL;
    SSafeStandstill : SAFEBOOL;
    SSafeMotionActive : SAFEBOOL;
    SFEmergencyStop1 : SFEmergencyStop;
    SFSafetyRequest1 : SFSafetyRequest;
    SFSafetyRequest2 : SFSafetyRequest;
    SFModeSelector1 : SFModeSelector;
    SFGuardLocking1 : SFGuardLocking;
    SFEnableSwitch1 : SFEnableSwitch;
END_VAR
VAR_OUTPUT
    SSafeStopM1 : SAFEBOOL;
    SSafeMotionM1 : SAFEBOOL;
    SEnableM1 : SAFEBOOL;
    SUnlockGuardK1 : SAFEBOOL;
END_VAR

SFEmergencyStop1(Activate:=TRUE, SEStopIn:=S1SEStopIn, SStartReset:=FALSE, SAutoReset:=FALSE, Reset:=S0Reset);
SFSafetyRequest1(Activate:=TRUE, SOpMode:=SFEmergencyStop1.SEStopOut, SAcknowledge:=M1SAcknowledgeSS1, MonitoringTime:=T#100ms, Reset:=S0Reset);
SFSafetyRequest2(Activate:=TRUE, SOpMode:=SAutoMode, SAcknowledge:=M1SAcknowledgeSafeMotion, MonitoringTime:=T#100ms, Reset:=S0Reset);
SFModeSelector1(Activate:=TRUE, SMode0:=S2SAutoMode, SMode1:=S2SSetupMode, SMode2:=FALSE, SMode3:=FALSE, SMode4:=FALSE, SMode5:=FALSE, SMode6:=FALSE, SMode7:=FALSE, SUnlock:=TRUE, SSetMode:=FALSE,
 AutoSetMode:=TRUE, ModeMonitorTime:=T#50ms, Reset:=S0Reset);
SFGuardLocking1(Activate:=TRUE, SGuardMonitoring:=S5SGuardSwitch, SSafetyActive:=SSafeStandstill OR SSafeMotionActive, SGuardLock:=S7SGuardLock, UnlockRequest:=S8UnlockGuard, SStartReset:=FALSE,
 SAutoReset:=FALSE, Reset:=S0Reset);
SFEnableSwitch1(Activate:=TRUE, SSafetyActive:=SSafeMotionActive AND SSetupMode, SEnableSwitchCh1:=S4SEnableSwitchCh1, SEnableSwitchCh2:=S4SEnableSwitchCh2, SAutoReset:=FALSE, Reset:=S0Reset);

SSafeStandstill := SFSafetyRequest1.SSafetyActive;
SSafeStopM1 := SFSafetyRequest1.SSafetyRequest;
SSafeMotionActive := SFSafetyRequest2.SSafetyActive;
SSafeMotionM1 := SFSafetyRequest2.SSafetyRequest;
SSetupMode := SFModeSelector1.SMode1Sel;
SAutoMode := SFModeSelector1.SMode0Sel AND SFGuardLocking1.SGuardLocked;
SUnlockGuardK1 := SFGuardLocking1.SUnlockGuard;
SEnableM1 := SFEnableSwitch1.SEnableSwitchOut;

END_PROGRAM

FUNCTION_BLOCK SFEmergencyStop
VAR_INPUT
    Activate : BOOL;
    SEStopIn : BOOL;
    SStartReset : BOOL;
    SAutoReset : BOOL;
    Reset : BOOL;
END_VAR
VAR
    RTRIGatReset : RTRIG;
END_VAR
VAR_OUTPUT
    Ready : BOOL;
    SEStopOut : BOOL;
    Error : BOOL;
    DiagCode : WORD;
END_VAR
RTRIGatReset(CLK:=Reset);
IF NOT Activate THEN
    DiagCode := 16#0000;
ELSE
    CASE DiagCode OF
    16#0000:
        IF Activate THEN
            DiagCode := 16#8001;
        END_IF;
    16#8001:
        IF NOT SStartReset THEN
            DiagCode := 16#8002;
        ELSIF SStartReset AND NOT SEStopIn THEN
            DiagCode := 16#8004;
        ELSIF SEStopIn AND SStartReset THEN
            DiagCode := 16#8000;
        END_IF;
    16#8002:
        IF SEStopIn THEN
            DiagCode := 16#8003;
        END_IF;
    16#8003:
        IF Reset AND NOT RTRIGatReset.Q THEN
            DiagCode := 16#C001;
        ELSIF NOT SEStopIn THEN
            DiagCode := 16#8002;
        ELSIF RTRIGatReset.Q THEN
            DiagCode := 16#8000;
        END_IF;
    16#C001:
        IF NOT Reset THEN
            DiagCode := 16#8003;
        END_IF;
    16#8004:
        IF SEStopIn AND NOT SAutoReset THEN
            DiagCode := 16#8005;
        ELSIF SEStopIn AND SAutoReset THEN
            DiagCode := 16#8000;
        END_IF;
    16#8005:
        IF Reset AND NOT RTRIGatReset.Q THEN
            DiagCode := 16#C002;
        ELSIF NOT SEStopIn THEN
            DiagCode := 16#8004;
        ELSIF RTRIGatReset.Q OR SAutoReset THEN
            DiagCode := 16#8000;
        END_IF;
    16#C002:
        IF NOT Reset THEN
            DiagCode := 16#8005;
        END_IF;
    16#8000:
        IF NOT SEStopIn THEN
            DiagCode := 16#8004;
        END_IF;
    END_CASE;
END_IF;
CASE DiagCode OF
16#0000:
    Ready := FALSE;
    Error := FALSE;
    SEStopOut := FALSE;
16#8001:
    Ready := TRUE;
    Error := FALSE;
    SEStopOut := FALSE;
16#8002:
    Ready := TRUE;
    Error := FALSE;
    SEStopOut := FALSE;
16#8003:
    Ready := TRUE;
    Error := FALSE;
    SEStopOut := FALSE;
16#C001:
    Ready := TRUE;
    Error := TRUE;
    SEStopOut := FALSE;
16#8004:
    Ready := TRUE;
    Error := FALSE;
    SEStopOut := FALSE;
16#8005:
    Ready := TRUE;
    Error := FALSE;
    SEStopOut := FALSE;
16#C002:
    Ready := TRUE;
    Error := TRUE;
    SEStopOut := FALSE;
16#8000:
    Ready := TRUE;
    Error := FALSE;
    SEStopOut := TRUE;
END_CASE;
END_FUNCTION_BLOCK

FUNCTION_BLOCK SFSafetyRequest
VAR_INPUT
    Activate : BOOL;
    SOpMode : SAFEBOOL;
    SAcknowledge : SAFEBOOL;
    MonitoringTime : TIME;
    Reset : BOOL;
END_VAR
VAR
    RTRIGatReset : RTRIG;
    Timer : TON;
END_VAR
VAR_OUTPUT
    Ready : BOOL;
    SSafetyActive : SAFEBOOL;
    SSafetyRequest : SAFEBOOL;
    Error : BOOL;
    DiagCode : WORD;
END_VAR
RTRIGatReset(CLK:=Reset);
IF NOT Activate THEN
    DiagCode := 16#0000;
ELSE
    CASE DiagCode OF
    16#0000:
        IF Activate THEN
            DiagCode := 16#8001;
        END_IF;
    16#8000:
        IF NOT SAcknowledge THEN
            DiagCode := 16#C002;
        ELSIF SOpMode THEN
            DiagCode := 16#8012;
        END_IF;
    16#8001:
        IF RTRIGatReset.Q AND NOT SAcknowledge THEN
            DiagCode := 16#8002;
        ELSIF RTRIGatReset.Q AND SAcknowledge THEN
            DiagCode := 16#8012;
        END_IF;
    16#8002:
        IF NOT SOpMode THEN
            DiagCode := 16#8003;
        ELSIF SAcknowledge THEN
            DiagCode := 16#8012;
        END_IF;
    16#8003:
        IF Timer.Q THEN
            DiagCode := 16#C003;
        ELSIF SOpMode THEN
            DiagCode := 16#8012;
        ELSIF SAcknowledge THEN
            DiagCode := 16#8000;
        END_IF;
    16#8005:
        IF SOpMode THEN
            DiagCode := 16#8012;
        END_IF;
    16#8012:
        IF NOT SAcknowledge THEN
            DiagCode := 16#8002;
        ELSIF NOT SOpMode THEN
            DiagCode := 16#8003;
        END_IF;
    16#C002:
        IF Reset AND NOT RTRIGatReset.Q THEN
            DiagCode := 16#C004;
        ELSIF RTRIGatReset.Q THEN
            DiagCode := 16#8005;
        END_IF;
    16#C003:
        IF Reset AND NOT RTRIGatReset.Q THEN
            DiagCode := 16#C005;
        ELSIF RTRIGatReset.Q THEN
            DiagCode := 16#8005;
        END_IF;
    16#C004:
        IF NOT Reset THEN
            DiagCode := 16#C002;
        END_IF;
    16#C005:
        IF NOT Reset THEN
            DiagCode := 16#C003;
        END_IF;
    END_CASE;
END_IF;
IF DiagCode <> 16#8003 THEN
    Timer(IN:=FALSE, PT:=MonitoringTime);
ELSE
    Timer(IN:=TRUE, PT:=MonitoringTime);
END_IF;
CASE DiagCode OF
16#0000:
    Ready := FALSE;
    SSafetyActive := FALSE;
    SSafetyRequest := FALSE;
    Error := FALSE;
16#8000:
    Ready := TRUE;
    SSafetyActive := TRUE;
    SSafetyRequest := FALSE;
    Error := FALSE;
16#8001:
    Ready := TRUE;
    SSafetyActive := FALSE;
    SSafetyRequest := FALSE;
    Error := FALSE;
16#8002:
    Ready := TRUE;
    SSafetyActive := FALSE;
    SSafetyRequest := TRUE;
    Error := FALSE;
16#8003:
    Ready := TRUE;
    SSafetyActive := FALSE;
    SSafetyRequest := FALSE;
    Error := FALSE;
16#8005:
    Ready := TRUE;
    SSafetyActive := FALSE;
    SSafetyRequest := FALSE;
    Error := FALSE;
16#8012:
    Ready := TRUE;
    SSafetyActive := FALSE;
    SSafetyRequest := TRUE;
    Error := FALSE;
16#C002:
    Ready := TRUE;
    SSafetyActive := FALSE;
    SSafetyRequest := FALSE;
    Error := TRUE;
16#C003:
    Ready := TRUE;
    SSafetyActive := FALSE;
    SSafetyRequest := FALSE;
    Error := TRUE;
16#C004:
    Ready := TRUE;
    SSafetyActive := FALSE;
    SSafetyRequest := FALSE;
    Error := TRUE;
16#C005:
    Ready := TRUE;
    SSafetyActive := FALSE;
    SSafetyRequest := FALSE;
    Error := TRUE;
END_CASE;
END_FUNCTION_BLOCK

FUNCTION_BLOCK SFModeSelector
VAR_INPUT
    Activate : BOOL;
    SMode0 : BOOL;
    SMode1 : BOOL;
    SMode2 : BOOL;
    SMode3 : BOOL;
    SMode4 : BOOL;
    SMode5 : BOOL;
    SMode6 : BOOL;
    SMode7 : BOOL;
    SUnlock : BOOL;
    SSetMode : BOOL;
    AutoSetMode : BOOL;
    ModeMonitorTime : TIME;
    Reset : BOOL;
END_VAR
VAR
    Timer : TON;
    RTRIGatReset: RTRIG;
    RTRIGatSetMode: RTRIG;
    FTRIGatModeSel0: FTRIG;
    RTRIGatModeSel0: RTRIG;
    fallingEdgeDetected : BOOL;
END_VAR
VAR_TEMP
    Error1 : BOOL;
    Error2 : BOOL;
END_VAR
VAR_OUTPUT
    Ready : BOOL;
    SMode0Sel : BOOL;
    SMode1Sel : BOOL;
    SMode2Sel : BOOL;
    SMode3Sel : BOOL;
    SMode4Sel : BOOL;
    SMode5Sel : BOOL;
    SMode6Sel : BOOL;
    SMode7Sel : BOOL;
    SAnyModeSel : BOOL;
    Error : BOOL;
    DiagCode : WORD;
END_VAR
RTRIGatReset(CLK:=Reset);
RTRIGatSetMode(CLK:=SSetMode);
IF NOT Activate THEN
    DiagCode := 16#0000;
ELSE
    IF (SMode0 + SMode1 + SMode2 + SMode3 + SMode4 + SMode5 + SMode6 + SMode7 > 1) THEN
        Error1 := true;
    ELSE
        Error1 := false;
    END_IF;
    CASE DiagCode OF
    16#0000:
        IF Activate THEN
            DiagCode := 16#8005;
        END_IF;
    16#8005:
        IF (NOT SMode0 AND NOT SMode1 AND NOT SMode2 AND NOT SMode3 AND NOT SMode4 AND NOT SMode5 AND NOT SMode6 AND NOT SMode7) THEN
            FTRIGatModeSel0(CLK:=false);
            RTRIGatModeSel0(CLK:=false);
        ELSE
            FTRIGatModeSel0(CLK:=true);
            RTRIGatModeSel0(CLK:=true);
        END_IF;
        IF FTRIGatModeSel0.Q THEN
            fallingEdgeDetected := TRUE;
        END_IF;
        IF fallingEdgeDetected THEN
            Timer(IN:=TRUE, PT:=ModeMonitorTime);
        ELSIF RTRIGatModeSel0.Q THEN
            Timer(IN:=FALSE, PT:=ModeMonitorTime);
            fallingEdgeDetected := FALSE;
        END_IF;
        Error2 := Timer.Q;
        IF Error1 THEN
            DiagCode := 16#C001;
        ELSIF Error2 THEN
            DiagCode := 16#C002;
        ELSIF ((AutoSetMode OR RTRIGatSetMode.Q) AND SUnlock AND (SMode0 + SMode1 + SMode2 + SMode3 + SMode4 + SMode5 + SMode6 + SMode7 = 1)) THEN
            DiagCode := 16#8000;
        END_IF;
    16#8000:
        IF Error1 THEN
            DiagCode := 16#C001;
        ELSIF (SMode0 <> SMode0Sel OR SMode1 <> SMode1Sel OR SMode2 <> SMode2Sel OR SMode3 <> SMode3Sel
              OR SMode4 <> SMode4Sel OR SMode5 <> SMode5Sel OR SMode6 <> SMode6Sel OR SMode7 <> SMode7Sel) THEN
            DiagCode := 16#8005;
            fallingEdgeDetected := FALSE;
        ELSIF (NOT SUnlock) THEN
            DiagCode := 16#8004;
        END_IF;
    16#8004:
        IF SUnlock THEN
            DiagCode := 16#8000;
        END_IF;
    16#C001:
        IF Reset AND NOT RTRIGatReset.Q THEN
            DiagCode := 16#C003;
        ELSIF RTRIGatReset.Q THEN
            DiagCode := 16#8005;
            fallingEdgeDetected := FALSE;
        END_IF;
    16#C002:
        IF Reset AND NOT RTRIGatReset.Q THEN
            DiagCode := 16#C004;
        ELSIF RTRIGatReset.Q THEN
            DiagCode := 16#8005;
            fallingEdgeDetected := FALSE;
        END_IF;
    16#C003:
        IF (NOT Reset) THEN
            DiagCode := 16#C001;
        END_IF;
    16#C004:
        IF (NOT Reset) THEN
            DiagCode := 16#C002;
        END_IF;
    END_CASE;
END_IF;

CASE DiagCode OF
16#0000:
    Ready := false;
    SMode0Sel := false;
    SMode1Sel := false;
    SMode2Sel := false;
    SMode3Sel := false;
    SMode4Sel := false;
    SMode5Sel := false;
    SMode6Sel := false;
    SMode7Sel := false;
    SAnyModeSel := false;
    Error := false;
16#8005:
    Ready := true;
    SMode0Sel := false;
    SMode1Sel := false;
    SMode2Sel := false;
    SMode3Sel := false;
    SMode4Sel := false;
    SMode5Sel := false;
    SMode6Sel := false;
    SMode7Sel := false;
    SAnyModeSel := false;
    Error := false;
16#8000:
    Ready := true;
    SMode0Sel := SMode0;
    SMode1Sel := SMode1;
    SMode2Sel := SMode2;
    SMode3Sel := SMode3;
    SMode4Sel := SMode4;
    SMode5Sel := SMode5;
    SMode6Sel := SMode6;
    SMode7Sel := SMode7;
    SAnyModeSel := true;
    Error := false;
16#8004:
    Ready := true;
    SAnyModeSel := true;
    Error := false;
16#C001,
16#C002,
16#C003,
16#C004:
    Ready := true;
    SMode0Sel := false;
    SMode1Sel := false;
    SMode2Sel := false;
    SMode3Sel := false;
    SMode4Sel := false;
    SMode5Sel := false;
    SMode6Sel := false;
    SMode7Sel := false;
    SAnyModeSel := false;
    Error := true;
END_CASE;
IF (DiagCode <> 16#8005) THEN
    Timer(IN:=FALSE, PT:=ModeMonitorTime);
END_IF;
END_FUNCTION_BLOCK

FUNCTION_BLOCK SFGuardLocking
VAR_INPUT
    Activate : BOOL;
    SGuardMonitoring : SAFEBOOL;
    SSafetyActive : SAFEBOOL;
    SGuardLock : SAFEBOOL;
    UnlockRequest : BOOL;
    SStartReset : SAFEBOOL;
    SAutoReset : SAFEBOOL;
    Reset : BOOL;
END_VAR
VAR
    RTRIGatReset : RTRIG;
    RTRIGatUnlockRequest : RTRIG;
END_VAR
VAR_OUTPUT
    Ready : BOOL;
    SGuardLocked : SAFEBOOL;
    SUnlockGuard : SAFEBOOL;
    Error : BOOL;
    DiagCode : WORD;
END_VAR
RTRIGatReset(CLK:=Reset);
RTRIGatUnlockRequest(CLK:=UnlockRequest);
IF NOT Activate THEN
    DiagCode := 16#0000;
END_IF;
CASE DiagCode OF
16#0000:
    IF Activate THEN
        DiagCode := 16#8001;
    END_IF;
16#8000:
    IF NOT SGuardLock OR NOT SGuardMonitoring THEN
        DiagCode := 16#C004;
    ELSIF RTRIGatUnlockRequest.Q AND SSafetyActive THEN
        DiagCode := 16#8013;
    END_IF;
16#8001:
    IF Reset AND NOT RTRIGatReset.Q AND NOT SStartReset THEN
        DiagCode := 16#C001;
    ELSIF NOT SGuardLock OR NOT SGuardMonitoring THEN
        DiagCode := 16#8011;
    ELSIF (RTRIGatReset.Q OR SStartReset) AND SGuardMonitoring AND SGuardLock THEN
        DiagCode := 16#8000;
    END_IF;
16#8003:
    IF Reset AND NOT RTRIGatReset.Q AND NOT SAutoReset THEN
        DiagCode := 16#C003;
    ELSIF NOT SGuardMonitoring OR NOT SGuardLock THEN
        DiagCode := 16#8011;
    ELSIF RTRIGatReset.Q OR SAutoReset THEN
        DiagCode := 16#8000;
    END_IF;
16#8011:
    IF NOT SSafetyActive AND (NOT SGuardMonitoring OR NOT SGuardLock) THEN
        DiagCode := 16#C004;
    ELSIF (SSafetyActive AND UnlockRequest) OR NOT SGuardMonitoring THEN
        DiagCode := 16#8012;
    ELSIF SGuardMonitoring AND SGuardLock THEN
        DiagCode := 16#8003;
    END_IF;
16#8012:
    IF SGuardMonitoring THEN
        DiagCode := 16#8013;
    ELSIF NOT SSafetyActive AND NOT SGuardMonitoring THEN
        DiagCode := 16#C004;
    END_IF;
16#8013:
    IF NOT SGuardMonitoring THEN
        DiagCode := 16#8012;
    ELSIF NOT UnlockRequest THEN
        DiagCode := 16#8011;
    END_IF;
16#8014:
    IF Reset AND NOT RTRIGatReset.Q THEN
        DiagCode := 16#C002;
    ELSIF NOT SSafetyActive THEN
        DiagCode := 16#C004;
    ELSIF RTRIGatReset.Q THEN
        DiagCode := 16#8011;
    END_IF;
16#C001:
    IF NOT Reset THEN
        DiagCode := 16#8001;
    END_IF;
16#C002:
    IF NOT Reset THEN
        DiagCode := 16#8014;
    END_IF;
16#C003:
    IF NOT Reset THEN
        DiagCode := 16#8003;
    END_IF;
16#C004:
    IF SSafetyActive THEN
        DiagCode := 16#8014;
    END_IF;
END_CASE;
CASE DiagCode OF
16#0000:
    Ready := FALSE;
    SGuardLocked := FALSE;
    SUnlockGuard := FALSE;
    Error := FALSE;
16#8000:
    Ready := TRUE;
    SGuardLocked := TRUE;
    SUnlockGuard := FALSE;
    Error := FALSE;
16#8001,
16#8003,
16#8011,
16#8014:
    Ready := TRUE;
    SGuardLocked := FALSE;
    SUnlockGuard := FALSE;
    Error := FALSE;
16#8012,
16#8013:
    Ready := TRUE;
    SGuardLocked := FALSE;
    SUnlockGuard := TRUE;
    Error := FALSE;
16#C001,
16#C002,
16#C003,
16#C004:
    Ready := TRUE;
    SGuardLocked := FALSE;
    SUnlockGuard := FALSE;
    Error := TRUE;
END_CASE;
END_FUNCTION_BLOCK

FUNCTION_BLOCK SFEnableSwitch
VAR_INPUT
    Activate : BOOL;
    SSafetyActive : SAFEBOOL;
    SEnableSwitchCh1 : SAFEBOOL;
    SEnableSwitchCh2 : SAFEBOOL;
    SAutoReset : SAFEBOOL;
    Reset : BOOL;
END_VAR
VAR
    RTRIGatReset : RTRIG;
END_VAR
VAR_OUTPUT
    Ready : BOOL;
    SEnableSwitchOut : SAFEBOOL;
    Error : BOOL;
    DiagCode : WORD;
END_VAR
RTRIGatReset(CLK:=Reset);
IF NOT Activate THEN
    DiagCode := 16#0000;
ELSIF NOT SSafetyActive THEN
    DiagCode := 16#8004;
ELSE
    CASE DiagCode OF
    16#0000:
        IF Activate THEN
            DiagCode := 16#8004;
        END_IF;
    16#8000:
        IF (NOT (SEnableSwitchCh1 OR SEnableSwitchCh2)) OR (SEnableSwitchCh1 AND NOT SEnableSwitchCh2) THEN
            DiagCode := 16#8007;
        ELSIF NOT SEnableSwitchCh1 AND SEnableSwitchCh2 THEN
            DiagCode := 16#8006;
        END_IF;
    16#8004:
        IF SSafetyActive THEN
            DiagCode := 16#8005;
        END_IF;
    16#8005:
        IF NOT (NOT SEnableSwitchCh1 AND SEnableSwitchCh2) THEN
            DiagCode := 16#C010;
        ELSIF NOT SEnableSwitchCh1 AND SEnableSwitchCh2 THEN
            DiagCode := 16#8006;
        END_IF;
    16#8006:
        IF SEnableSwitchCh1 AND SEnableSwitchCh2 THEN
            DiagCode := 16#8000;
        ELSIF (NOT (SEnableSwitchCh1 OR SEnableSwitchCh2)) OR (SEnableSwitchCh1 AND NOT SEnableSwitchCh2) THEN
            DiagCode := 16#8007;
        END_IF;
    16#8007:
        IF SEnableSwitchCh1 AND SEnableSwitchCh2 THEN
            DiagCode := 16#C030;
        ELSIF NOT SEnableSwitchCh1 AND SEnableSwitchCh2 THEN
            DiagCode := 16#8006;
        END_IF;
    16#C001:
        IF NOT Reset THEN
            DiagCode := 16#C020;
        END_IF;
    16#C002:
        IF NOT Reset THEN
            DiagCode := 16#C040;
        END_IF;
    16#C010:
        IF NOT SEnableSwitchCh1 AND SEnableSwitchCh2 THEN
            DiagCode := 16#C020;
        END_IF;
    16#C020:
        IF NOT (NOT SEnableSwitchCh1 AND SEnableSwitchCh2) THEN
            DiagCode := 16#C010;
        ELSIF Reset AND NOT RTRIGatReset.Q AND NOT SAutoReset THEN
            DiagCode := 16#C001;
        ELSIF RTRIGatReset.Q OR SAutoReset THEN
            DiagCode := 16#8006;
        END_IF;
    16#C030:
        IF NOT (SEnableSwitchCh1 AND SEnableSwitchCh2) THEN
            DiagCode := 16#C040;
        END_IF;
    16#C040:
        IF SEnableSwitchCh1 AND SEnableSwitchCh2 THEN
            DiagCode := 16#C030;
        ELSIF Reset AND RTRIGatReset.Q AND NOT SAutoReset THEN
            DiagCode := 16#C002;
        ELSIF RTRIGatReset.Q OR SAutoReset THEN
            DiagCode := 16#8007;
        END_IF;
    END_CASE;
END_IF;

CASE DiagCode OF
16#C001,
16#C002,
16#C010,
16#C020,
16#C030,
16#C040:
    Ready := TRUE;
    SEnableSwitchOut := FALSE;
    Error := TRUE;
16#0000:
    Ready := FALSE;
    SEnableSwitchOut := FALSE;
    Error := FALSE;
16#8000:
    Ready := TRUE;
    SEnableSwitchOut := TRUE;
    Error := FALSE;
16#8004,
16#8005,
16#8006,
16#8007:
    Ready := TRUE;
    SEnableSwitchOut := FALSE;
    Error := FALSE;
END_CASE;
END_FUNCTION_BLOCK

FUNCTION_BLOCK RTRIG
VAR_INPUT
    CLK : BOOL;
END_VAR
VAR
    M : BOOL;
END_VAR
VAR_OUTPUT
    Q : BOOL;
END_VAR
    Q := CLK AND NOT M;
    M := CLK;
END_FUNCTION_BLOCK

FUNCTION_BLOCK TON
VAR_INPUT
    IN : BOOL;
    PT : TIME;
END_VAR
VAR
    running : BOOL;
END_VAR
VAR_TEMP
    timeout : BOOL;
END_VAR
VAR_OUTPUT
    Q : BOOL;
    ET : TIME;
END_VAR
timeout := NONDETERMINISTIC_BOOL();
IF NOT IN THEN
    Q := FALSE;
    running := FALSE;
ELSIF NOT running AND NOT Q THEN
    running := TRUE;
ELSIF running AND NOT Q THEN
    Q := timeout;
    running := NOT Q;
END_IF;
ET := NONDETERMINISTIC_TIME();
END_FUNCTION_BLOCK

FUNCTION_BLOCK FTRIG
VAR_INPUT
    CLK : BOOL;
END_VAR
VAR
   M : BOOL;
END_VAR
VAR_OUTPUT
   Q : BOOL;
END_VAR
    Q := NOT CLK AND M;
    M := CLK;
END_FUNCTION_BLOCK
